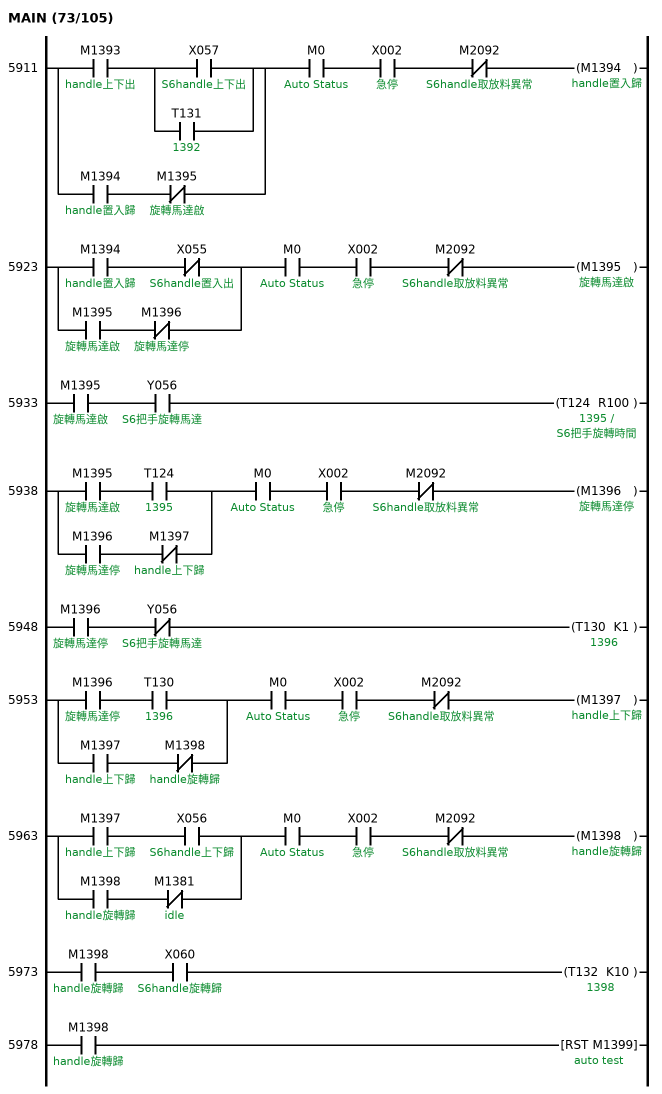
[picture p72: ladder of MAIN, rungs at steps 5911 to 5978]
5911  LD      M1393  ; handle上下出
      LD      X057  ; S6handle上下出
      OR      T131  ; 1392
      ANB
      LD      M1394  ; handle置入歸
      ANI     M1395  ; 旋轉馬達啟
      ORB
      AND     M0  ; Auto Status
      AND     X002  ; 急停
      ANI     M2092  ; S6handle取放料異常
      OUT     M1394  ; handle置入歸
5923  LD      M1394  ; handle置入歸
      ANI     X055  ; S6handle置入出
      LD      M1395  ; 旋轉馬達啟
      ANI     M1396  ; 旋轉馬達停
      ORB
      AND     M0  ; Auto Status
      AND     X002  ; 急停
      ANI     M2092  ; S6handle取放料異常
      OUT     M1395  ; 旋轉馬達啟
5933  LD      M1395  ; 旋轉馬達啟
      AND     Y056  ; S6把手旋轉馬達
      OUT     T124 R100  ; 1395 / S6把手旋轉時間
5938  LD      M1395  ; 旋轉馬達啟
      AND     T124  ; 1395
      LD      M1396  ; 旋轉馬達停
      ANI     M1397  ; handle上下歸
      ORB
      AND     M0  ; Auto Status
      AND     X002  ; 急停
      ANI     M2092  ; S6handle取放料異常
      OUT     M1396  ; 旋轉馬達停
5948  LD      M1396  ; 旋轉馬達停
      ANI     Y056  ; S6把手旋轉馬達
      OUT     T130 K1  ; 1396
5953  LD      M1396  ; 旋轉馬達停
      AND     T130  ; 1396
      LD      M1397  ; handle上下歸
      ANI     M1398  ; handle旋轉歸
      ORB
      AND     M0  ; Auto Status
      AND     X002  ; 急停
      ANI     M2092  ; S6handle取放料異常
      OUT     M1397  ; handle上下歸
5963  LD      M1397  ; handle上下歸
      AND     X056  ; S6handle上下歸
      LD      M1398  ; handle旋轉歸
      ANI     M1381  ; idle
      ORB
      AND     M0  ; Auto Status
      AND     X002  ; 急停
      ANI     M2092  ; S6handle取放料異常
      OUT     M1398  ; handle旋轉歸
5973  LD      M1398  ; handle旋轉歸
      AND     X060  ; S6handle旋轉歸
      OUT     T132 K10  ; 1398
5978  LD      M1398  ; handle旋轉歸
      RST     M1399  ; auto test
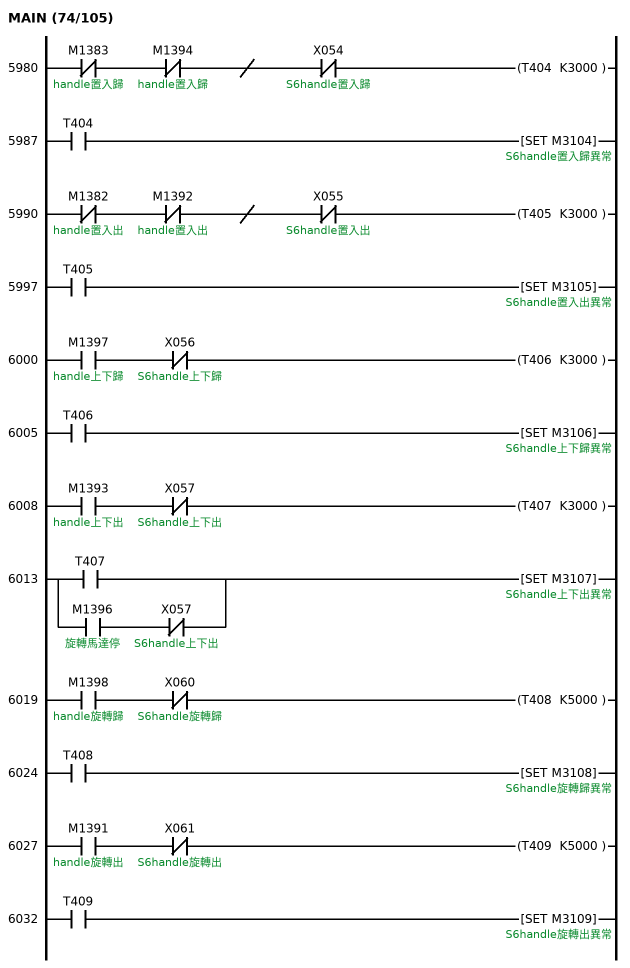
5980  LDI     M1383  ; handle置入歸
      ANI     M1394  ; handle置入歸
      INV
      ANI     X054  ; S6handle置入歸
      OUT     T404 K3000
5987  LD      T404
      SET     M3104  ; S6handle置入歸異常
5990  LDI     M1382  ; handle置入出
      ANI     M1392  ; handle置入出
      INV
      ANI     X055  ; S6handle置入出
      OUT     T405 K3000
5997  LD      T405
      SET     M3105  ; S6handle置入出異常
6000  LD      M1397  ; handle上下歸
      ANI     X056  ; S6handle上下歸
      OUT     T406 K3000
6005  LD      T406
      SET     M3106  ; S6handle上下歸異常
6008  LD      M1393  ; handle上下出
      ANI     X057  ; S6handle上下出
      OUT     T407 K3000
6013  LD      T407
      LD      M1396  ; 旋轉馬達停
      ANI     X057  ; S6handle上下出
      ORB
      SET     M3107  ; S6handle上下出異常
6019  LD      M1398  ; handle旋轉歸
      ANI     X060  ; S6handle旋轉歸
      OUT     T408 K5000
6024  LD      T408
      SET     M3108  ; S6handle旋轉歸異常
6027  LD      M1391  ; handle旋轉出
      ANI     X061  ; S6handle旋轉出
      OUT     T409 K5000
6032  LD      T409
      SET     M3109  ; S6handle旋轉出異常
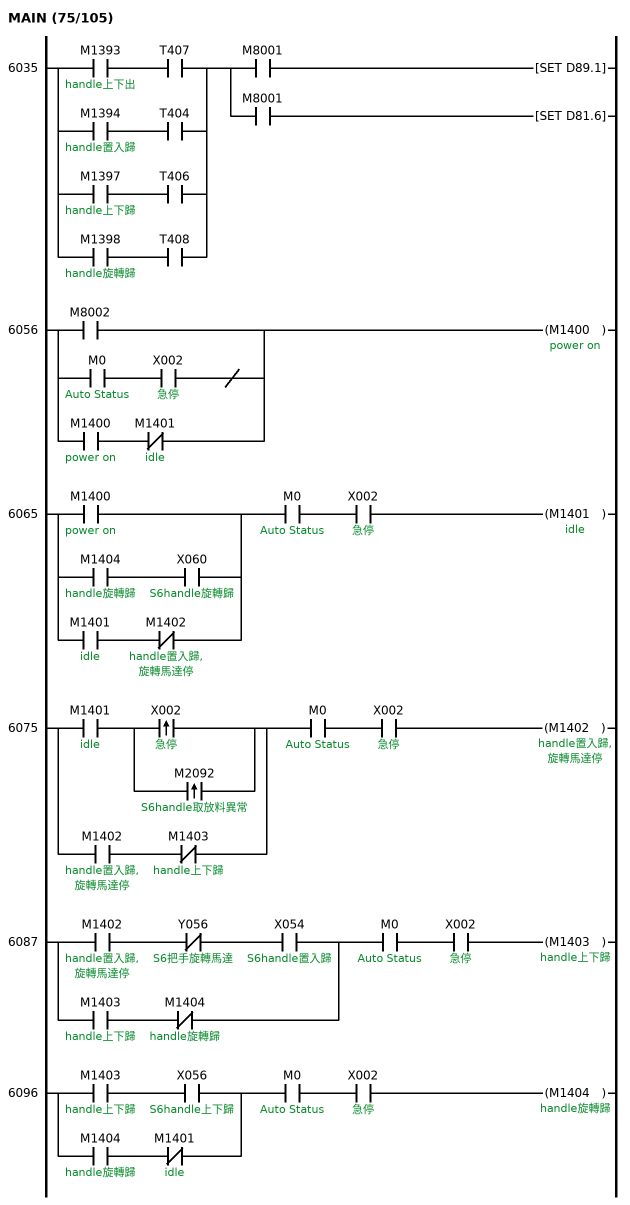
6035  LD      M1393  ; handle上下出
      AND     T407
      LD      M1394  ; handle置入歸
      AND     T404
      ORB
      LD      M1397  ; handle上下歸
      AND     T406
      ORB
      LD      M1398  ; handle旋轉歸
      AND     T408
      ORB
      MPS
      AND     M8001
      SET     D89.1
      MPP
      AND     M8001
      SET     D81.6
6056  LD      M8002
      LD      M0  ; Auto Status
      AND     X002  ; 急停
      INV
      ORB
      LD      M1400  ; power on
      ANI     M1401  ; idle
      ORB
      OUT     M1400  ; power on
6065  LD      M1400  ; power on
      LD      M1404  ; handle旋轉歸
      AND     X060  ; S6handle旋轉歸
      ORB
      LD      M1401  ; idle
      ANI     M1402  ; handle置入歸,旋轉馬達停
      ORB
      AND     M0  ; Auto Status
      AND     X002  ; 急停
      OUT     M1401  ; idle
6075  LD      M1401  ; idle
      LDP     X002  ; 急停
      ORP     M2092  ; S6handle取放料異常
      ANB
      LD      M1402  ; handle置入歸,旋轉馬達停
      ANI     M1403  ; handle上下歸
      ORB
      AND     M0  ; Auto Status
      AND     X002  ; 急停
      OUT     M1402  ; handle置入歸,旋轉馬達停
6087  LD      M1402  ; handle置入歸,旋轉馬達停
      ANI     Y056  ; S6把手旋轉馬達
      AND     X054  ; S6handle置入歸
      LD      M1403  ; handle上下歸
      ANI     M1404  ; handle旋轉歸
      ORB
      AND     M0  ; Auto Status
      AND     X002  ; 急停
      OUT     M1403  ; handle上下歸
6096  LD      M1403  ; handle上下歸
      AND     X056  ; S6handle上下歸
      LD      M1404  ; handle旋轉歸
      ANI     M1401  ; idle
      ORB
      AND     M0  ; Auto Status
      AND     X002  ; 急停
      OUT     M1404  ; handle旋轉歸
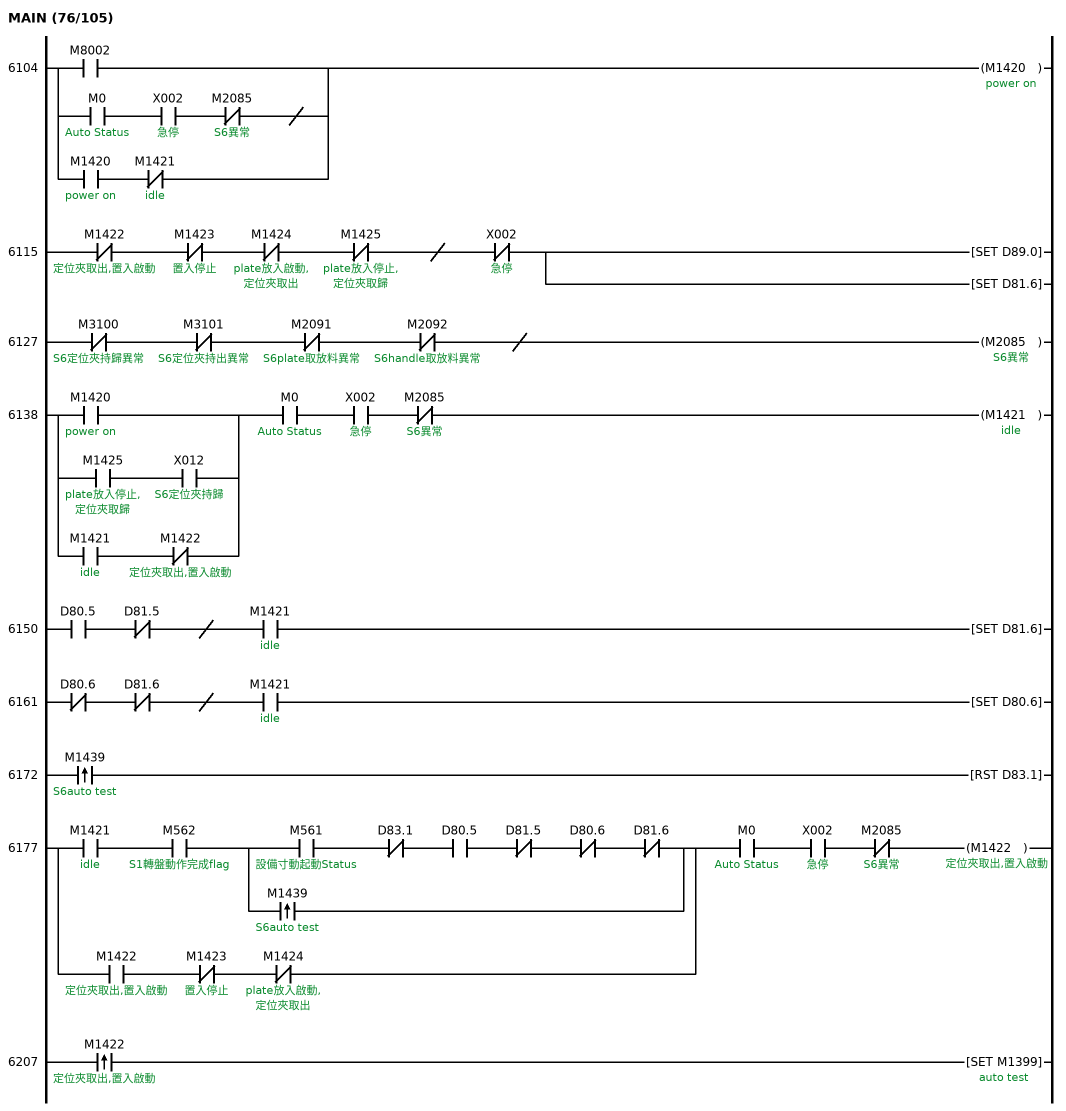
6104  LD      M8002
      LD      M0  ; Auto Status
      AND     X002  ; 急停
      ANI     M2085  ; S6異常
      INV
      ORB
      LD      M1420  ; power on
      ANI     M1421  ; idle
      ORB
      OUT     M1420  ; power on
6115  LDI     M1422  ; 定位夾取出,置入啟動
      ANI     M1423  ; 置入停止
      ANI     M1424  ; plate放入啟動,定位夾取出
      ANI     M1425  ; plate放入停止,定位夾取歸
      INV
      ANI     X002  ; 急停
      SET     D89.0
      SET     D81.6
6127  LDI     M3100  ; S6定位夾持歸異常
      ANI     M3101  ; S6定位夾持出異常
      ANI     M2091  ; S6plate取放料異常
      ANI     M2092  ; S6handle取放料異常
      INV
      OUT     M2085  ; S6異常
6138  LD      M1420  ; power on
      LD      M1425  ; plate放入停止,定位夾取歸
      AND     X012  ; S6定位夾持歸
      ORB
      LD      M1421  ; idle
      ANI     M1422  ; 定位夾取出,置入啟動
      ORB
      AND     M0  ; Auto Status
      AND     X002  ; 急停
      ANI     M2085  ; S6異常
      OUT     M1421  ; idle
6150  LD      D80.5
      ANI     D81.5
      INV
      AND     M1421  ; idle
      SET     D81.6
6161  LDI     D80.6
      ANI     D81.6
      INV
      AND     M1421  ; idle
      SET     D80.6
6172  LDP     M1439  ; S6auto test
      RST     D83.1
6177  LD      M1421  ; idle
      AND     M562  ; S1轉盤動作完成flag
      LD      M561  ; 設備寸動起動Status
      ANI     D83.1
      AND     D80.5
      ANI     D81.5
      ANI     D80.6
      ANI     D81.6
      ORP     M1439  ; S6auto test
      ANB
      LD      M1422  ; 定位夾取出,置入啟動
      ANI     M1423  ; 置入停止
      ANI     M1424  ; plate放入啟動,定位夾取出
      ORB
      AND     M0  ; Auto Status
      AND     X002  ; 急停
      ANI     M2085  ; S6異常
      OUT     M1422  ; 定位夾取出,置入啟動
6207  LDP     M1422  ; 定位夾取出,置入啟動
      SET     M1399  ; auto test
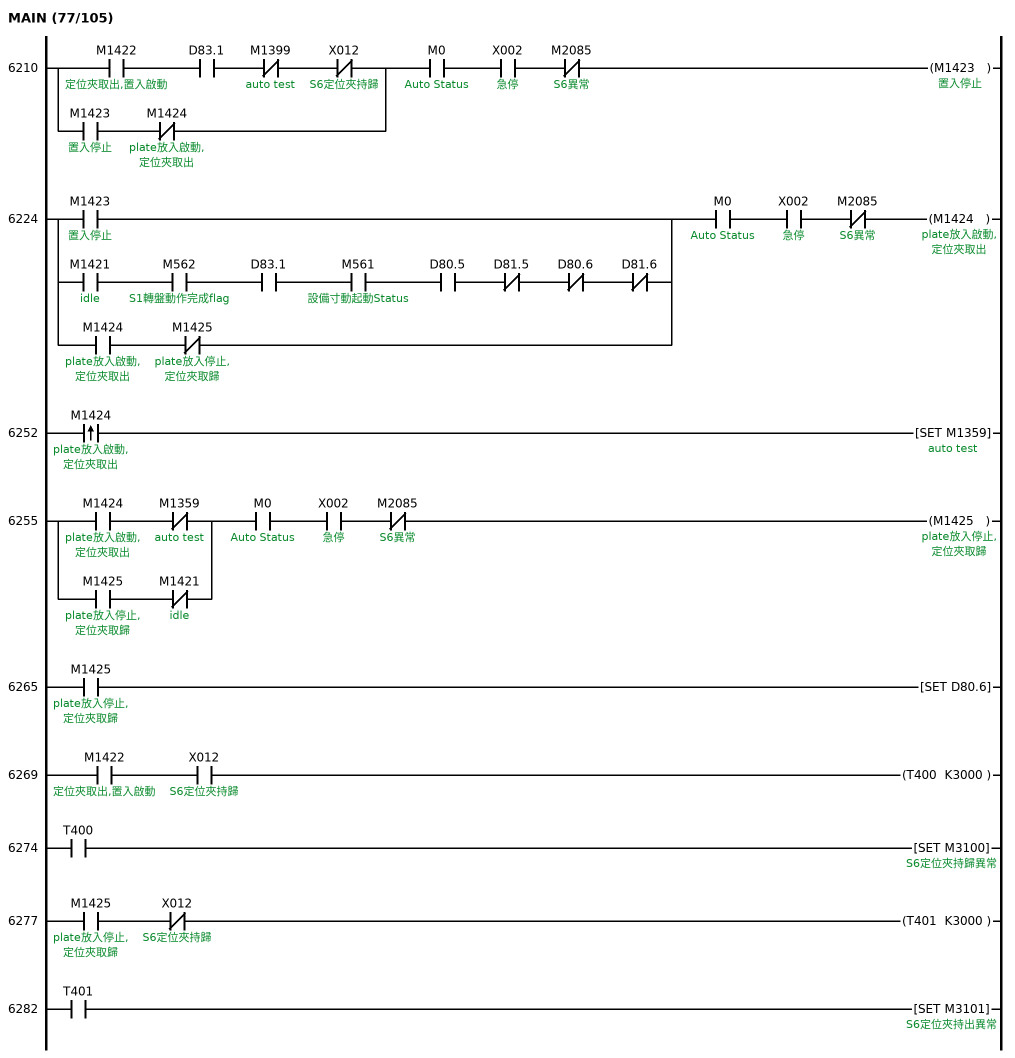
6210  LD      M1422  ; 定位夾取出,置入啟動
      AND     D83.1
      ANI     M1399  ; auto test
      ANI     X012  ; S6定位夾持歸
      LD      M1423  ; 置入停止
      ANI     M1424  ; plate放入啟動,定位夾取出
      ORB
      AND     M0  ; Auto Status
      AND     X002  ; 急停
      ANI     M2085  ; S6異常
      OUT     M1423  ; 置入停止
6224  LD      M1423  ; 置入停止
      LD      M1421  ; idle
      AND     M562  ; S1轉盤動作完成flag
      AND     D83.1
      AND     M561  ; 設備寸動起動Status
      AND     D80.5
      ANI     D81.5
      ANI     D80.6
      ANI     D81.6
      ORB
      LD      M1424  ; plate放入啟動,定位夾取出
      ANI     M1425  ; plate放入停止,定位夾取歸
      ORB
      AND     M0  ; Auto Status
      AND     X002  ; 急停
      ANI     M2085  ; S6異常
      OUT     M1424  ; plate放入啟動,定位夾取出
6252  LDP     M1424  ; plate放入啟動,定位夾取出
      SET     M1359  ; auto test
6255  LD      M1424  ; plate放入啟動,定位夾取出
      ANI     M1359  ; auto test
      LD      M1425  ; plate放入停止,定位夾取歸
      ANI     M1421  ; idle
      ORB
      AND     M0  ; Auto Status
      AND     X002  ; 急停
      ANI     M2085  ; S6異常
      OUT     M1425  ; plate放入停止,定位夾取歸
6265  LD      M1425  ; plate放入停止,定位夾取歸
      SET     D80.6
6269  LD      M1422  ; 定位夾取出,置入啟動
      AND     X012  ; S6定位夾持歸
      OUT     T400 K3000
6274  LD      T400
      SET     M3100  ; S6定位夾持歸異常
6277  LD      M1425  ; plate放入停止,定位夾取歸
      ANI     X012  ; S6定位夾持歸
      OUT     T401 K3000
6282  LD      T401
      SET     M3101  ; S6定位夾持出異常
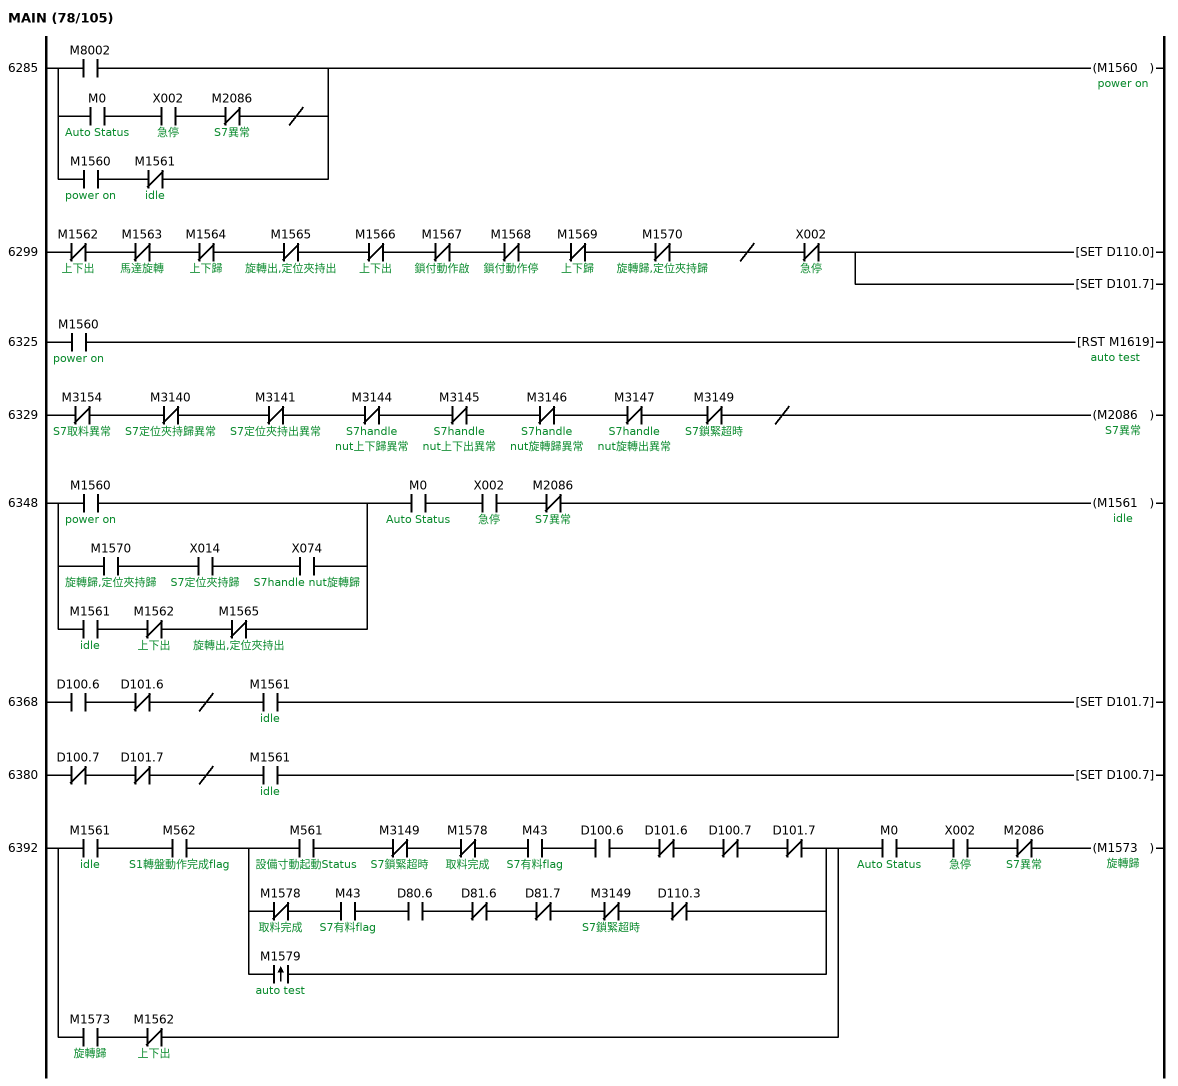
6285  LD      M8002
      LD      M0  ; Auto Status
      AND     X002  ; 急停
      ANI     M2086  ; S7異常
      INV
      ORB
      LD      M1560  ; power on
      ANI     M1561  ; idle
      ORB
      OUT     M1560  ; power on
6299  LDI     M1562  ; 上下出
      ANI     M1563  ; 馬達旋轉
      ANI     M1564  ; 上下歸
      ANI     M1565  ; 旋轉出,定位夾持出
      ANI     M1566  ; 上下出
      ANI     M1567  ; 鎖付動作啟
      ANI     M1568  ; 鎖付動作停
      ANI     M1569  ; 上下歸
      ANI     M1570  ; 旋轉歸,定位夾持歸
      INV
      ANI     X002  ; 急停
      SET     D110.0
      SET     D101.7
6325  LD      M1560  ; power on
      RST     M1619  ; auto test
6329  LDI     M3154  ; S7取料異常
      ANI     M3140  ; S7定位夾持歸異常
      ANI     M3141  ; S7定位夾持出異常
      ANI     M3144  ; S7handle nut上下歸異常
      ANI     M3145  ; S7handle nut上下出異常
      ANI     M3146  ; S7handle nut旋轉歸異常
      ANI     M3147  ; S7handle nut旋轉出異常
      ANI     M3149  ; S7鎖緊超時
      INV
      OUT     M2086  ; S7異常
6348  LD      M1560  ; power on
      LD      M1570  ; 旋轉歸,定位夾持歸
      AND     X014  ; S7定位夾持歸
      AND     X074  ; S7handle nut旋轉歸
      ORB
      LD      M1561  ; idle
      ANI     M1562  ; 上下出
      ANI     M1565  ; 旋轉出,定位夾持出
      ORB
      AND     M0  ; Auto Status
      AND     X002  ; 急停
      ANI     M2086  ; S7異常
      OUT     M1561  ; idle
6368  LD      D100.6
      ANI     D101.6
      INV
      AND     M1561  ; idle
      SET     D101.7
6380  LDI     D100.7
      ANI     D101.7
      INV
      AND     M1561  ; idle
      SET     D100.7
6392  LD      M1561  ; idle
      AND     M562  ; S1轉盤動作完成flag
      LD      M561  ; 設備寸動起動Status
      ANI     M3149  ; S7鎖緊超時
      ANI     M1578  ; 取料完成
      AND     M43  ; S7有料flag
      AND     D100.6
      ANI     D101.6
      ANI     D100.7
      ANI     D101.7
      LDI     M1578  ; 取料完成
      AND     M43  ; S7有料flag
      AND     D80.6
      ANI     D81.6
      ANI     D81.7
      ANI     M3149  ; S7鎖緊超時
      ANI     D110.3
      ORB
      ORP     M1579  ; auto test
      ANB
      LD      M1573  ; 旋轉歸
      ANI     M1562  ; 上下出
      ORB
      AND     M0  ; Auto Status
      AND     X002  ; 急停
      ANI     M2086  ; S7異常
      OUT     M1573  ; 旋轉歸
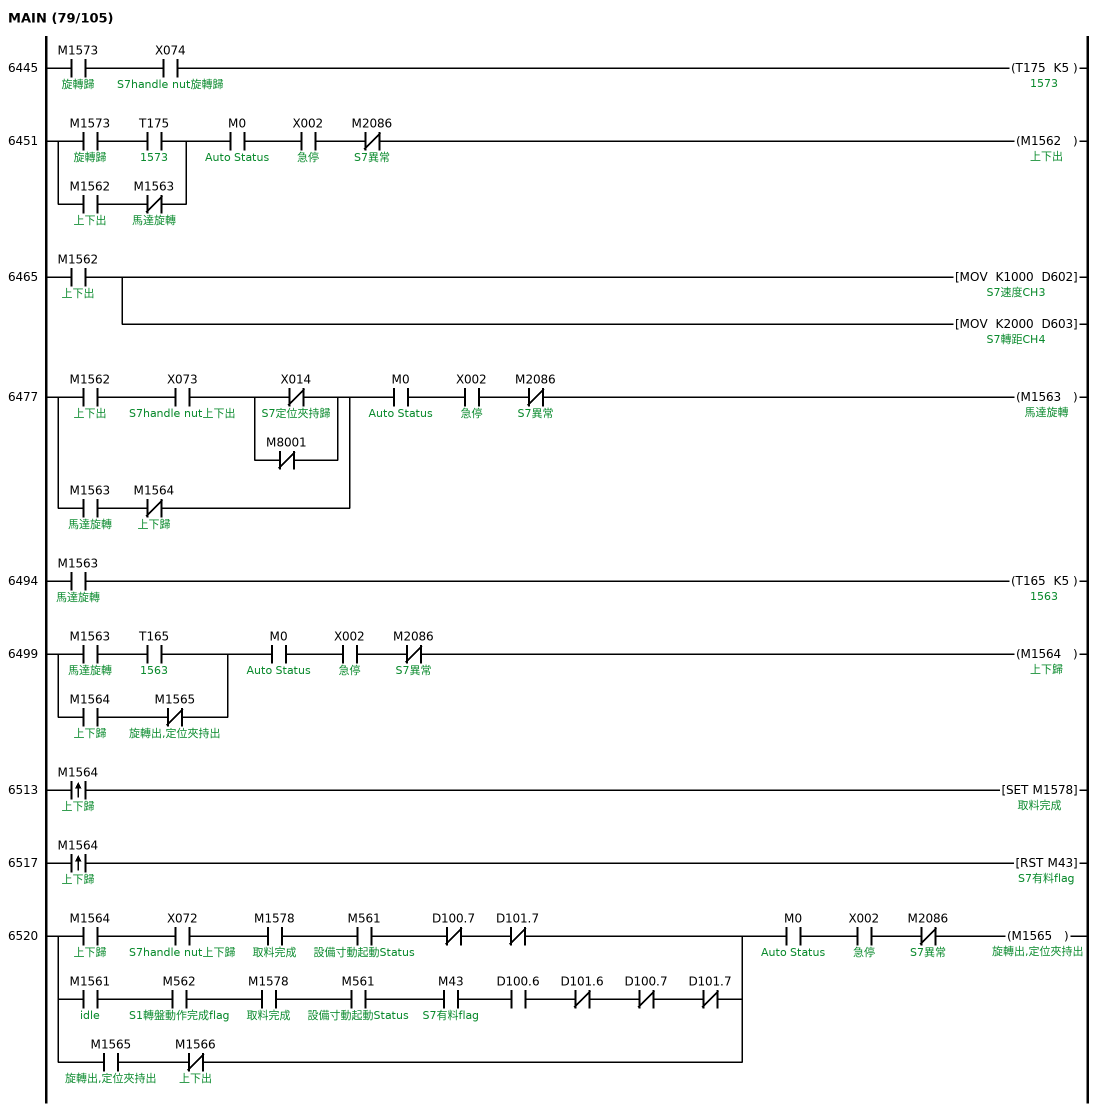
6445  LD      M1573  ; 旋轉歸
      AND     X074  ; S7handle nut旋轉歸
      OUT     T175 K5  ; 1573
6451  LD      M1573  ; 旋轉歸
      AND     T175  ; 1573
      LD      M1562  ; 上下出
      ANI     M1563  ; 馬達旋轉
      ORB
      AND     M0  ; Auto Status
      AND     X002  ; 急停
      ANI     M2086  ; S7異常
      OUT     M1562  ; 上下出
6465  LD      M1562  ; 上下出
      MOV     K1000 D602  ; S7速度CH3
      MOV     K2000 D603  ; S7轉距CH4
6477  LD      M1562  ; 上下出
      AND     X073  ; S7handle nut上下出
      LDI     X014  ; S7定位夾持歸
      ORI     M8001
      ANB
      LD      M1563  ; 馬達旋轉
      ANI     M1564  ; 上下歸
      ORB
      AND     M0  ; Auto Status
      AND     X002  ; 急停
      ANI     M2086  ; S7異常
      OUT     M1563  ; 馬達旋轉
6494  LD      M1563  ; 馬達旋轉
      OUT     T165 K5  ; 1563
6499  LD      M1563  ; 馬達旋轉
      AND     T165  ; 1563
      LD      M1564  ; 上下歸
      ANI     M1565  ; 旋轉出,定位夾持出
      ORB
      AND     M0  ; Auto Status
      AND     X002  ; 急停
      ANI     M2086  ; S7異常
      OUT     M1564  ; 上下歸
6513  LDP     M1564  ; 上下歸
      SET     M1578  ; 取料完成
6517  LDP     M1564  ; 上下歸
      RST     M43  ; S7有料flag
6520  LD      M1564  ; 上下歸
      AND     X072  ; S7handle nut上下歸
      AND     M1578  ; 取料完成
      AND     M561  ; 設備寸動起動Status
      ANI     D100.7
      ANI     D101.7
      LD      M1561  ; idle
      AND     M562  ; S1轉盤動作完成flag
      AND     M1578  ; 取料完成
      AND     M561  ; 設備寸動起動Status
      AND     M43  ; S7有料flag
      AND     D100.6
      ANI     D101.6
      ANI     D100.7
      ANI     D101.7
      ORB
      LD      M1565  ; 旋轉出,定位夾持出
      ANI     M1566  ; 上下出
      ORB
      AND     M0  ; Auto Status
      AND     X002  ; 急停
      ANI     M2086  ; S7異常
      OUT     M1565  ; 旋轉出,定位夾持出
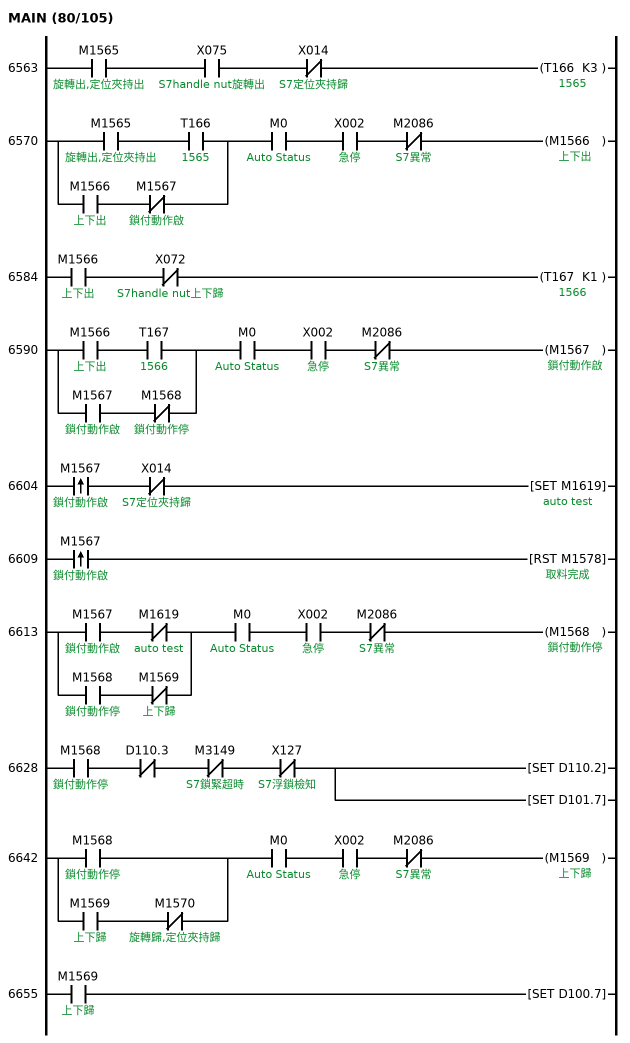
6563  LD      M1565  ; 旋轉出,定位夾持出
      AND     X075  ; S7handle nut旋轉出
      ANI     X014  ; S7定位夾持歸
      OUT     T166 K3  ; 1565
6570  LD      M1565  ; 旋轉出,定位夾持出
      AND     T166  ; 1565
      LD      M1566  ; 上下出
      ANI     M1567  ; 鎖付動作啟
      ORB
      AND     M0  ; Auto Status
      AND     X002  ; 急停
      ANI     M2086  ; S7異常
      OUT     M1566  ; 上下出
6584  LD      M1566  ; 上下出
      ANI     X072  ; S7handle nut上下歸
      OUT     T167 K1  ; 1566
6590  LD      M1566  ; 上下出
      AND     T167  ; 1566
      LD      M1567  ; 鎖付動作啟
      ANI     M1568  ; 鎖付動作停
      ORB
      AND     M0  ; Auto Status
      AND     X002  ; 急停
      ANI     M2086  ; S7異常
      OUT     M1567  ; 鎖付動作啟
6604  LDP     M1567  ; 鎖付動作啟
      ANI     X014  ; S7定位夾持歸
      SET     M1619  ; auto test
6609  LDP     M1567  ; 鎖付動作啟
      RST     M1578  ; 取料完成
6613  LD      M1567  ; 鎖付動作啟
      ANI     M1619  ; auto test
      LD      M1568  ; 鎖付動作停
      ANI     M1569  ; 上下歸
      ORB
      AND     M0  ; Auto Status
      AND     X002  ; 急停
      ANI     M2086  ; S7異常
      OUT     M1568  ; 鎖付動作停
6628  LD      M1568  ; 鎖付動作停
      ANI     D110.3
      ANI     M3149  ; S7鎖緊超時
      ANI     X127  ; S7浮鎖檢知
      SET     D110.2
      SET     D101.7
6642  LD      M1568  ; 鎖付動作停
      LD      M1569  ; 上下歸
      ANI     M1570  ; 旋轉歸,定位夾持歸
      ORB
      AND     M0  ; Auto Status
      AND     X002  ; 急停
      ANI     M2086  ; S7異常
      OUT     M1569  ; 上下歸
6655  LD      M1569  ; 上下歸
      SET     D100.7
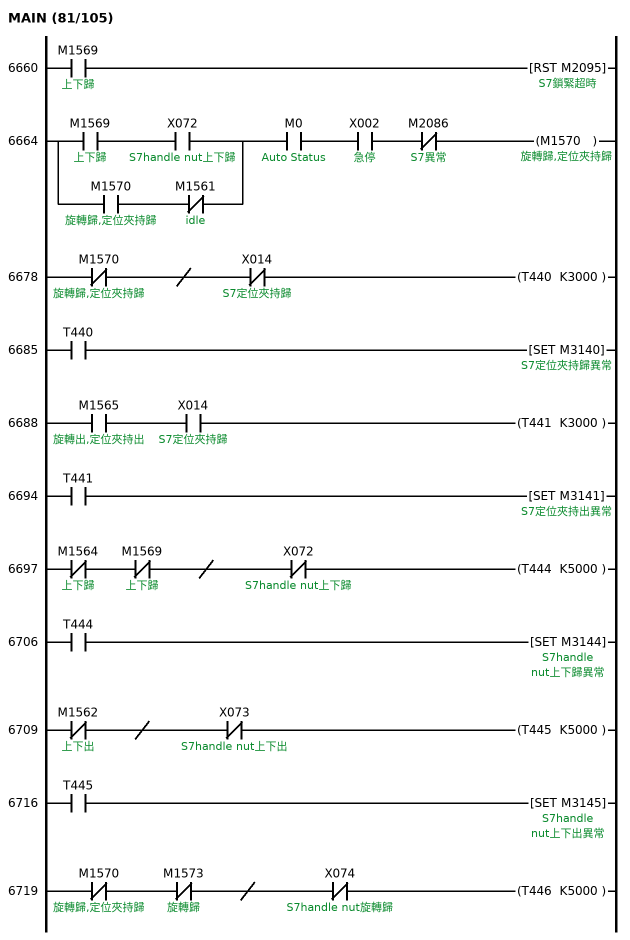
6660  LD      M1569  ; 上下歸
      RST     M2095  ; S7鎖緊超時
6664  LD      M1569  ; 上下歸
      AND     X072  ; S7handle nut上下歸
      LD      M1570  ; 旋轉歸,定位夾持歸
      ANI     M1561  ; idle
      ORB
      AND     M0  ; Auto Status
      AND     X002  ; 急停
      ANI     M2086  ; S7異常
      OUT     M1570  ; 旋轉歸,定位夾持歸
6678  LDI     M1570  ; 旋轉歸,定位夾持歸
      INV
      ANI     X014  ; S7定位夾持歸
      OUT     T440 K3000
6685  LD      T440
      SET     M3140  ; S7定位夾持歸異常
6688  LD      M1565  ; 旋轉出,定位夾持出
      AND     X014  ; S7定位夾持歸
      OUT     T441 K3000
6694  LD      T441
      SET     M3141  ; S7定位夾持出異常
6697  LDI     M1564  ; 上下歸
      ANI     M1569  ; 上下歸
      INV
      ANI     X072  ; S7handle nut上下歸
      OUT     T444 K5000
6706  LD      T444
      SET     M3144  ; S7handle nut上下歸異常
6709  LDI     M1562  ; 上下出
      INV
      ANI     X073  ; S7handle nut上下出
      OUT     T445 K5000
6716  LD      T445
      SET     M3145  ; S7handle nut上下出異常
6719  LDI     M1570  ; 旋轉歸,定位夾持歸
      ANI     M1573  ; 旋轉歸
      INV
      ANI     X074  ; S7handle nut旋轉歸
      OUT     T446 K5000
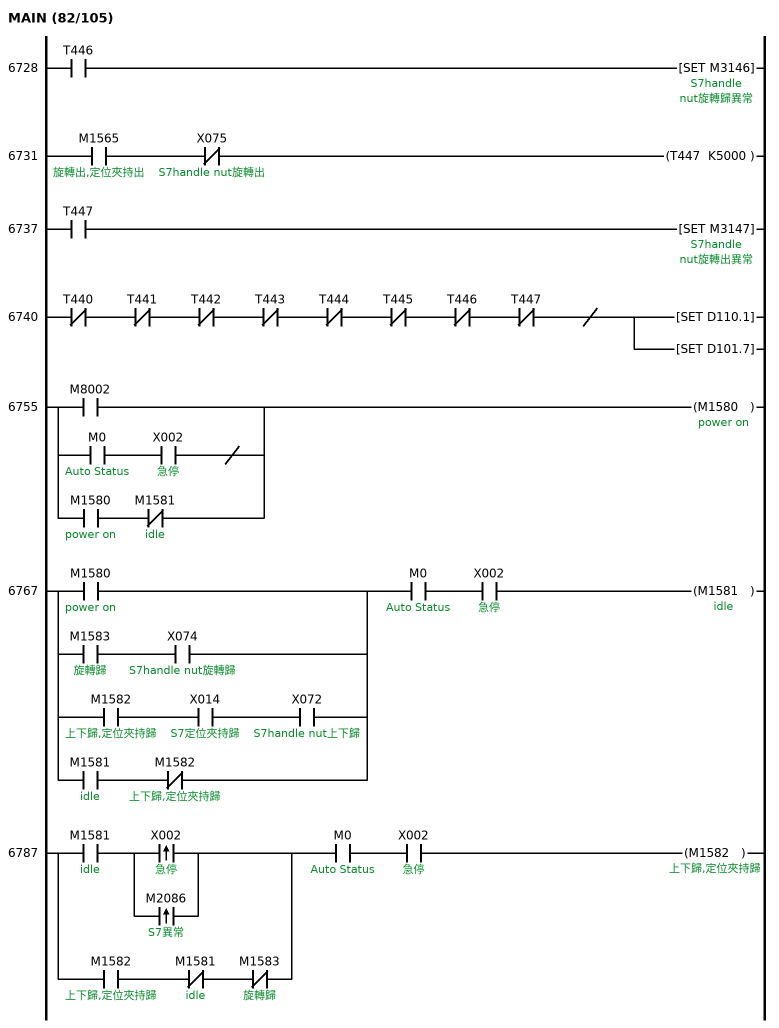
6728  LD      T446
      SET     M3146  ; S7handle nut旋轉歸異常
6731  LD      M1565  ; 旋轉出,定位夾持出
      ANI     X075  ; S7handle nut旋轉出
      OUT     T447 K5000
6737  LD      T447
      SET     M3147  ; S7handle nut旋轉出異常
6740  LDI     T440
      ANI     T441
      ANI     T442
      ANI     T443
      ANI     T444
      ANI     T445
      ANI     T446
      ANI     T447
      INV
      SET     D110.1
      SET     D101.7
6755  LD      M8002
      LD      M0  ; Auto Status
      AND     X002  ; 急停
      INV
      ORB
      LD      M1580  ; power on
      ANI     M1581  ; idle
      ORB
      OUT     M1580  ; power on
6767  LD      M1580  ; power on
      LD      M1583  ; 旋轉歸
      AND     X074  ; S7handle nut旋轉歸
      ORB
      LD      M1582  ; 上下歸,定位夾持歸
      AND     X014  ; S7定位夾持歸
      AND     X072  ; S7handle nut上下歸
      ORB
      LD      M1581  ; idle
      ANI     M1582  ; 上下歸,定位夾持歸
      ORB
      AND     M0  ; Auto Status
      AND     X002  ; 急停
      OUT     M1581  ; idle
6787  LD      M1581  ; idle
      LDP     X002  ; 急停
      ORP     M2086  ; S7異常
      ANB
      LD      M1582  ; 上下歸,定位夾持歸
      ANI     M1581  ; idle
      ANI     M1583  ; 旋轉歸
      ORB
      AND     M0  ; Auto Status
      AND     X002  ; 急停
      OUT     M1582  ; 上下歸,定位夾持歸
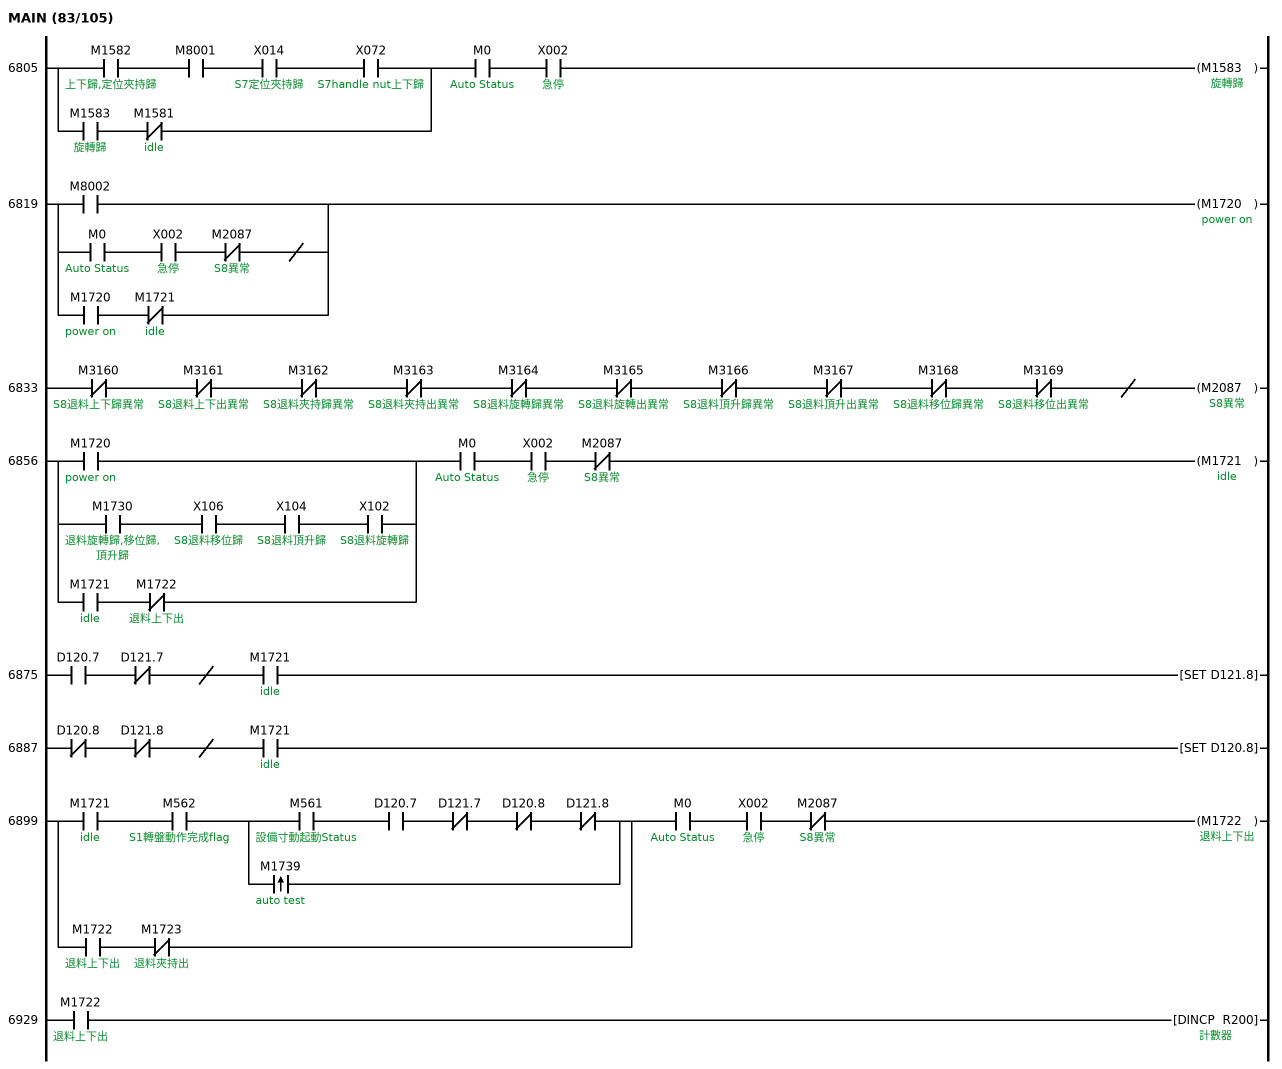
6805  LD      M1582  ; 上下歸,定位夾持歸
      AND     M8001
      AND     X014  ; S7定位夾持歸
      AND     X072  ; S7handle nut上下歸
      LD      M1583  ; 旋轉歸
      ANI     M1581  ; idle
      ORB
      AND     M0  ; Auto Status
      AND     X002  ; 急停
      OUT     M1583  ; 旋轉歸
6819  LD      M8002
      LD      M0  ; Auto Status
      AND     X002  ; 急停
      ANI     M2087  ; S8異常
      INV
      ORB
      LD      M1720  ; power on
      ANI     M1721  ; idle
      ORB
      OUT     M1720  ; power on
6833  LDI     M3160  ; S8退料上下歸異常
      ANI     M3161  ; S8退料上下出異常
      ANI     M3162  ; S8退料夾持歸異常
      ANI     M3163  ; S8退料夾持出異常
      ANI     M3164  ; S8退料旋轉歸異常
      ANI     M3165  ; S8退料旋轉出異常
      ANI     M3166  ; S8退料頂升歸異常
      ANI     M3167  ; S8退料頂升出異常
      ANI     M3168  ; S8退料移位歸異常
      ANI     M3169  ; S8退料移位出異常
      INV
      OUT     M2087  ; S8異常
6856  LD      M1720  ; power on
      LD      M1730  ; 退料旋轉歸,移位歸,頂升歸
      AND     X106  ; S8退料移位歸
      AND     X104  ; S8退料頂升歸
      AND     X102  ; S8退料旋轉歸
      ORB
      LD      M1721  ; idle
      ANI     M1722  ; 退料上下出
      ORB
      AND     M0  ; Auto Status
      AND     X002  ; 急停
      ANI     M2087  ; S8異常
      OUT     M1721  ; idle
6875  LD      D120.7
      ANI     D121.7
      INV
      AND     M1721  ; idle
      SET     D121.8
6887  LDI     D120.8
      ANI     D121.8
      INV
      AND     M1721  ; idle
      SET     D120.8
6899  LD      M1721  ; idle
      AND     M562  ; S1轉盤動作完成flag
      LD      M561  ; 設備寸動起動Status
      AND     D120.7
      ANI     D121.7
      ANI     D120.8
      ANI     D121.8
      ORP     M1739  ; auto test
      ANB
      LD      M1722  ; 退料上下出
      ANI     M1723  ; 退料夾持出
      ORB
      AND     M0  ; Auto Status
      AND     X002  ; 急停
      ANI     M2087  ; S8異常
      OUT     M1722  ; 退料上下出
6929  LD      M1722  ; 退料上下出
      DINCP   R200  ; 計數器
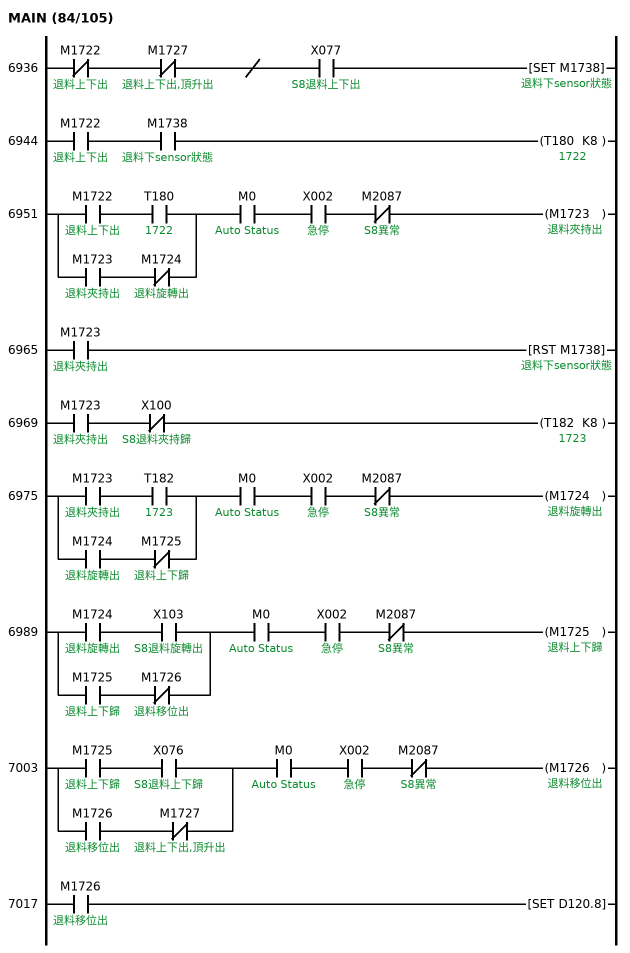
6936  LDI     M1722  ; 退料上下出
      ANI     M1727  ; 退料上下出,頂升出
      INV
      AND     X077  ; S8退料上下出
      SET     M1738  ; 退料下sensor狀態
6944  LD      M1722  ; 退料上下出
      AND     M1738  ; 退料下sensor狀態
      OUT     T180 K8  ; 1722
6951  LD      M1722  ; 退料上下出
      AND     T180  ; 1722
      LD      M1723  ; 退料夾持出
      ANI     M1724  ; 退料旋轉出
      ORB
      AND     M0  ; Auto Status
      AND     X002  ; 急停
      ANI     M2087  ; S8異常
      OUT     M1723  ; 退料夾持出
6965  LD      M1723  ; 退料夾持出
      RST     M1738  ; 退料下sensor狀態
6969  LD      M1723  ; 退料夾持出
      ANI     X100  ; S8退料夾持歸
      OUT     T182 K8  ; 1723
6975  LD      M1723  ; 退料夾持出
      AND     T182  ; 1723
      LD      M1724  ; 退料旋轉出
      ANI     M1725  ; 退料上下歸
      ORB
      AND     M0  ; Auto Status
      AND     X002  ; 急停
      ANI     M2087  ; S8異常
      OUT     M1724  ; 退料旋轉出
6989  LD      M1724  ; 退料旋轉出
      AND     X103  ; S8退料旋轉出
      LD      M1725  ; 退料上下歸
      ANI     M1726  ; 退料移位出
      ORB
      AND     M0  ; Auto Status
      AND     X002  ; 急停
      ANI     M2087  ; S8異常
      OUT     M1725  ; 退料上下歸
7003  LD      M1725  ; 退料上下歸
      AND     X076  ; S8退料上下歸
      LD      M1726  ; 退料移位出
      ANI     M1727  ; 退料上下出,頂升出
      ORB
      AND     M0  ; Auto Status
      AND     X002  ; 急停
      ANI     M2087  ; S8異常
      OUT     M1726  ; 退料移位出
7017  LD      M1726  ; 退料移位出
      SET     D120.8
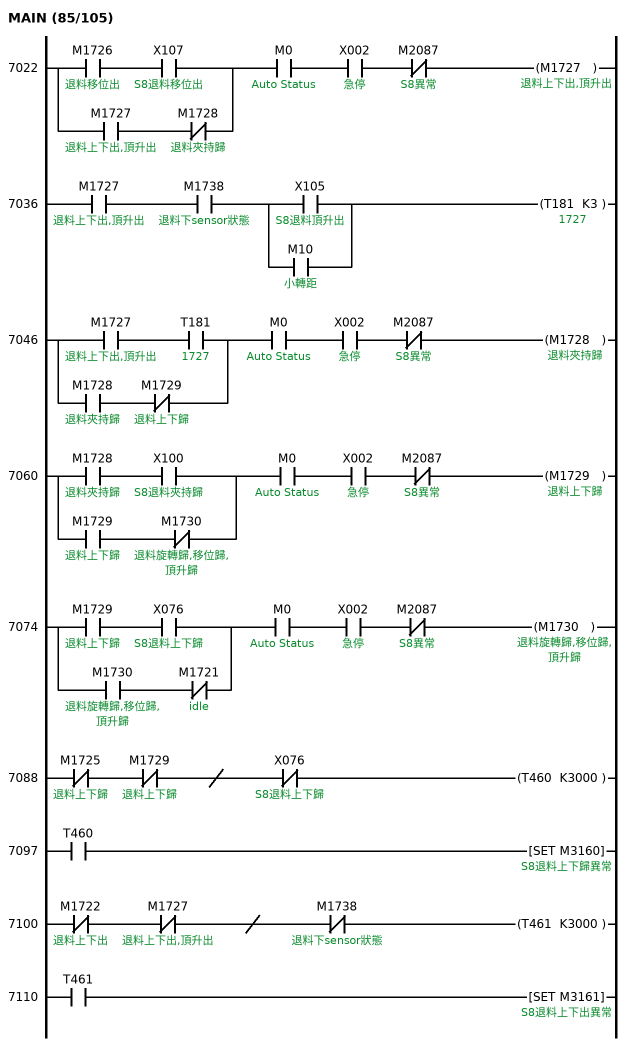
7022  LD      M1726  ; 退料移位出
      AND     X107  ; S8退料移位出
      LD      M1727  ; 退料上下出,頂升出
      ANI     M1728  ; 退料夾持歸
      ORB
      AND     M0  ; Auto Status
      AND     X002  ; 急停
      ANI     M2087  ; S8異常
      OUT     M1727  ; 退料上下出,頂升出
7036  LD      M1727  ; 退料上下出,頂升出
      AND     M1738  ; 退料下sensor狀態
      LD      X105  ; S8退料頂升出
      OR      M10  ; 小轉距
      ANB
      OUT     T181 K3  ; 1727
7046  LD      M1727  ; 退料上下出,頂升出
      AND     T181  ; 1727
      LD      M1728  ; 退料夾持歸
      ANI     M1729  ; 退料上下歸
      ORB
      AND     M0  ; Auto Status
      AND     X002  ; 急停
      ANI     M2087  ; S8異常
      OUT     M1728  ; 退料夾持歸
7060  LD      M1728  ; 退料夾持歸
      AND     X100  ; S8退料夾持歸
      LD      M1729  ; 退料上下歸
      ANI     M1730  ; 退料旋轉歸,移位歸,頂升歸
      ORB
      AND     M0  ; Auto Status
      AND     X002  ; 急停
      ANI     M2087  ; S8異常
      OUT     M1729  ; 退料上下歸
7074  LD      M1729  ; 退料上下歸
      AND     X076  ; S8退料上下歸
      LD      M1730  ; 退料旋轉歸,移位歸,頂升歸
      ANI     M1721  ; idle
      ORB
      AND     M0  ; Auto Status
      AND     X002  ; 急停
      ANI     M2087  ; S8異常
      OUT     M1730  ; 退料旋轉歸,移位歸,頂升歸
7088  LDI     M1725  ; 退料上下歸
      ANI     M1729  ; 退料上下歸
      INV
      ANI     X076  ; S8退料上下歸
      OUT     T460 K3000
7097  LD      T460
      SET     M3160  ; S8退料上下歸異常
7100  LDI     M1722  ; 退料上下出
      ANI     M1727  ; 退料上下出,頂升出
      INV
      ANI     M1738  ; 退料下sensor狀態
      OUT     T461 K3000
7110  LD      T461
      SET     M3161  ; S8退料上下出異常
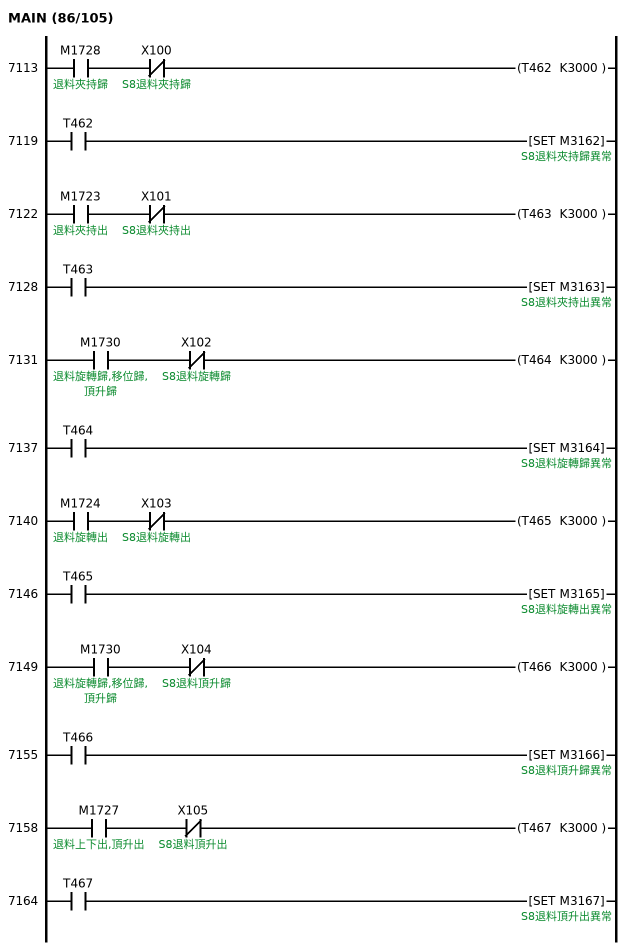
7113  LD      M1728  ; 退料夾持歸
      ANI     X100  ; S8退料夾持歸
      OUT     T462 K3000
7119  LD      T462
      SET     M3162  ; S8退料夾持歸異常
7122  LD      M1723  ; 退料夾持出
      ANI     X101  ; S8退料夾持出
      OUT     T463 K3000
7128  LD      T463
      SET     M3163  ; S8退料夾持出異常
7131  LD      M1730  ; 退料旋轉歸,移位歸,頂升歸
      ANI     X102  ; S8退料旋轉歸
      OUT     T464 K3000
7137  LD      T464
      SET     M3164  ; S8退料旋轉歸異常
7140  LD      M1724  ; 退料旋轉出
      ANI     X103  ; S8退料旋轉出
      OUT     T465 K3000
7146  LD      T465
      SET     M3165  ; S8退料旋轉出異常
7149  LD      M1730  ; 退料旋轉歸,移位歸,頂升歸
      ANI     X104  ; S8退料頂升歸
      OUT     T466 K3000
7155  LD      T466
      SET     M3166  ; S8退料頂升歸異常
7158  LD      M1727  ; 退料上下出,頂升出
      ANI     X105  ; S8退料頂升出
      OUT     T467 K3000
7164  LD      T467
      SET     M3167  ; S8退料頂升出異常
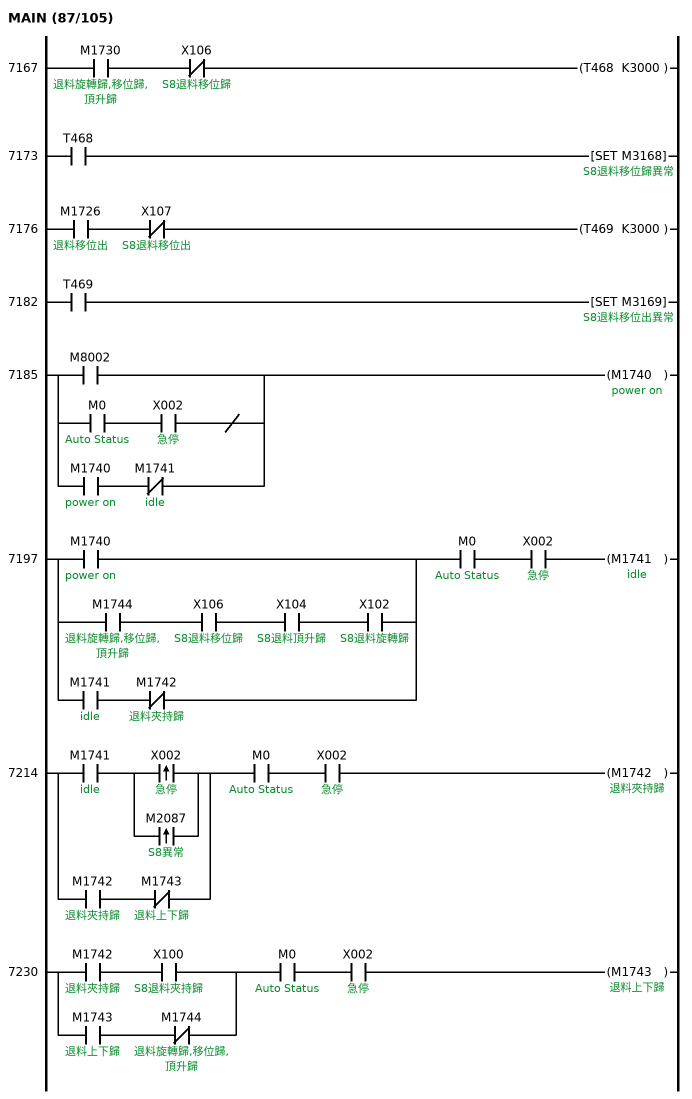
7167  LD      M1730  ; 退料旋轉歸,移位歸,頂升歸
      ANI     X106  ; S8退料移位歸
      OUT     T468 K3000
7173  LD      T468
      SET     M3168  ; S8退料移位歸異常
7176  LD      M1726  ; 退料移位出
      ANI     X107  ; S8退料移位出
      OUT     T469 K3000
7182  LD      T469
      SET     M3169  ; S8退料移位出異常
7185  LD      M8002
      LD      M0  ; Auto Status
      AND     X002  ; 急停
      INV
      ORB
      LD      M1740  ; power on
      ANI     M1741  ; idle
      ORB
      OUT     M1740  ; power on
7197  LD      M1740  ; power on
      LD      M1744  ; 退料旋轉歸,移位歸,頂升歸
      AND     X106  ; S8退料移位歸
      AND     X104  ; S8退料頂升歸
      AND     X102  ; S8退料旋轉歸
      ORB
      LD      M1741  ; idle
      ANI     M1742  ; 退料夾持歸
      ORB
      AND     M0  ; Auto Status
      AND     X002  ; 急停
      OUT     M1741  ; idle
7214  LD      M1741  ; idle
      LDP     X002  ; 急停
      ORP     M2087  ; S8異常
      ANB
      LD      M1742  ; 退料夾持歸
      ANI     M1743  ; 退料上下歸
      ORB
      AND     M0  ; Auto Status
      AND     X002  ; 急停
      OUT     M1742  ; 退料夾持歸
7230  LD      M1742  ; 退料夾持歸
      AND     X100  ; S8退料夾持歸
      LD      M1743  ; 退料上下歸
      ANI     M1744  ; 退料旋轉歸,移位歸,頂升歸
      ORB
      AND     M0  ; Auto Status
      AND     X002  ; 急停
      OUT     M1743  ; 退料上下歸
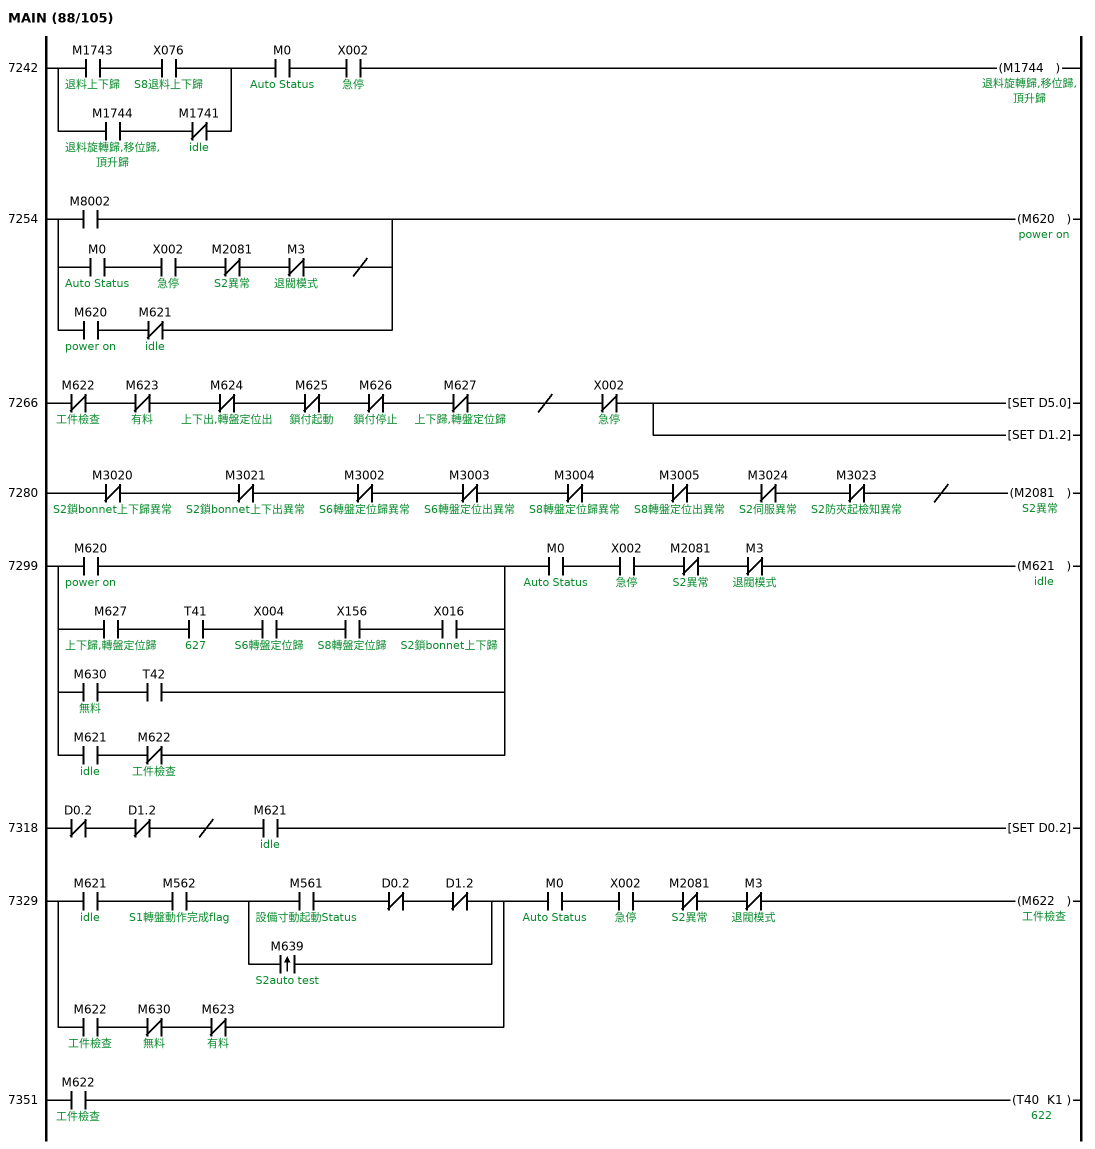
7242  LD      M1743  ; 退料上下歸
      AND     X076  ; S8退料上下歸
      LD      M1744  ; 退料旋轉歸,移位歸,頂升歸
      ANI     M1741  ; idle
      ORB
      AND     M0  ; Auto Status
      AND     X002  ; 急停
      OUT     M1744  ; 退料旋轉歸,移位歸,頂升歸
7254  LD      M8002
      LD      M0  ; Auto Status
      AND     X002  ; 急停
      ANI     M2081  ; S2異常
      ANI     M3  ; 退閥模式
      INV
      ORB
      LD      M620  ; power on
      ANI     M621  ; idle
      ORB
      OUT     M620  ; power on
7266  LDI     M622  ; 工件檢查
      ANI     M623  ; 有料
      ANI     M624  ; 上下出,轉盤定位出
      ANI     M625  ; 鎖付起動
      ANI     M626  ; 鎖付停止
      ANI     M627  ; 上下歸,轉盤定位歸
      INV
      ANI     X002  ; 急停
      SET     D5.0
      SET     D1.2
7280  LDI     M3020  ; S2鎖bonnet上下歸異常
      ANI     M3021  ; S2鎖bonnet上下出異常
      ANI     M3002  ; S6轉盤定位歸異常
      ANI     M3003  ; S6轉盤定位出異常
      ANI     M3004  ; S8轉盤定位歸異常
      ANI     M3005  ; S8轉盤定位出異常
      ANI     M3024  ; S2伺服異常
      ANI     M3023  ; S2防夾起檢知異常
      INV
      OUT     M2081  ; S2異常
7299  LD      M620  ; power on
      LD      M627  ; 上下歸,轉盤定位歸
      AND     T41  ; 627
      AND     X004  ; S6轉盤定位歸
      AND     X156  ; S8轉盤定位歸
      AND     X016  ; S2鎖bonnet上下歸
      ORB
      LD      M630  ; 無料
      AND     T42
      ORB
      LD      M621  ; idle
      ANI     M622  ; 工件檢查
      ORB
      AND     M0  ; Auto Status
      AND     X002  ; 急停
      ANI     M2081  ; S2異常
      ANI     M3  ; 退閥模式
      OUT     M621  ; idle
7318  LDI     D0.2
      ANI     D1.2
      INV
      AND     M621  ; idle
      SET     D0.2
7329  LD      M621  ; idle
      AND     M562  ; S1轉盤動作完成flag
      LD      M561  ; 設備寸動起動Status
      ANI     D0.2
      ANI     D1.2
      ORP     M639  ; S2auto test
      ANB
      LD      M622  ; 工件檢查
      ANI     M630  ; 無料
      ANI     M623  ; 有料
      ORB
      AND     M0  ; Auto Status
      AND     X002  ; 急停
      ANI     M2081  ; S2異常
      ANI     M3  ; 退閥模式
      OUT     M622  ; 工件檢查
7351  LD      M622  ; 工件檢查
      OUT     T40 K1  ; 622
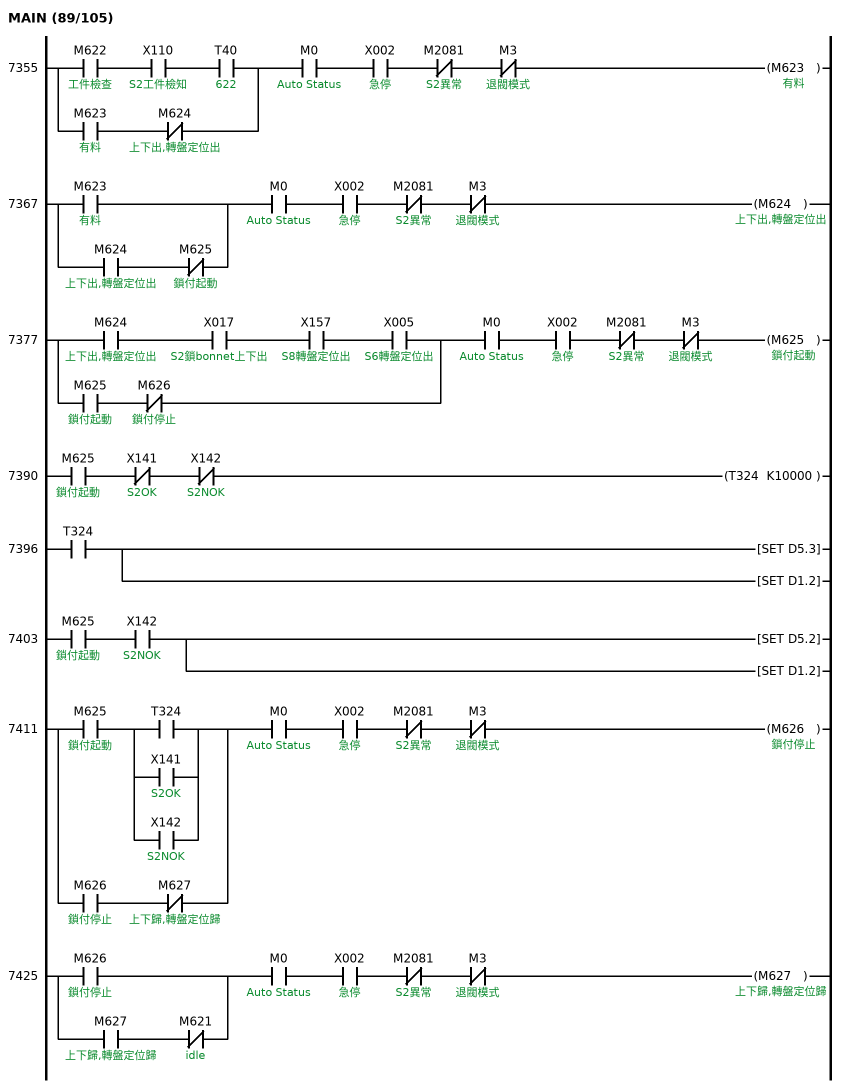
7355  LD      M622  ; 工件檢查
      AND     X110  ; S2工件檢知
      AND     T40  ; 622
      LD      M623  ; 有料
      ANI     M624  ; 上下出,轉盤定位出
      ORB
      AND     M0  ; Auto Status
      AND     X002  ; 急停
      ANI     M2081  ; S2異常
      ANI     M3  ; 退閥模式
      OUT     M623  ; 有料
7367  LD      M623  ; 有料
      LD      M624  ; 上下出,轉盤定位出
      ANI     M625  ; 鎖付起動
      ORB
      AND     M0  ; Auto Status
      AND     X002  ; 急停
      ANI     M2081  ; S2異常
      ANI     M3  ; 退閥模式
      OUT     M624  ; 上下出,轉盤定位出
7377  LD      M624  ; 上下出,轉盤定位出
      AND     X017  ; S2鎖bonnet上下出
      AND     X157  ; S8轉盤定位出
      AND     X005  ; S6轉盤定位出
      LD      M625  ; 鎖付起動
      ANI     M626  ; 鎖付停止
      ORB
      AND     M0  ; Auto Status
      AND     X002  ; 急停
      ANI     M2081  ; S2異常
      ANI     M3  ; 退閥模式
      OUT     M625  ; 鎖付起動
7390  LD      M625  ; 鎖付起動
      ANI     X141  ; S2OK
      ANI     X142  ; S2NOK
      OUT     T324 K10000
7396  LD      T324
      SET     D5.3
      SET     D1.2
7403  LD      M625  ; 鎖付起動
      AND     X142  ; S2NOK
      SET     D5.2
      SET     D1.2
7411  LD      M625  ; 鎖付起動
      LD      T324
      OR      X141  ; S2OK
      OR      X142  ; S2NOK
      ANB
      LD      M626  ; 鎖付停止
      ANI     M627  ; 上下歸,轉盤定位歸
      ORB
      AND     M0  ; Auto Status
      AND     X002  ; 急停
      ANI     M2081  ; S2異常
      ANI     M3  ; 退閥模式
      OUT     M626  ; 鎖付停止
7425  LD      M626  ; 鎖付停止
      LD      M627  ; 上下歸,轉盤定位歸
      ANI     M621  ; idle
      ORB
      AND     M0  ; Auto Status
      AND     X002  ; 急停
      ANI     M2081  ; S2異常
      ANI     M3  ; 退閥模式
      OUT     M627  ; 上下歸,轉盤定位歸
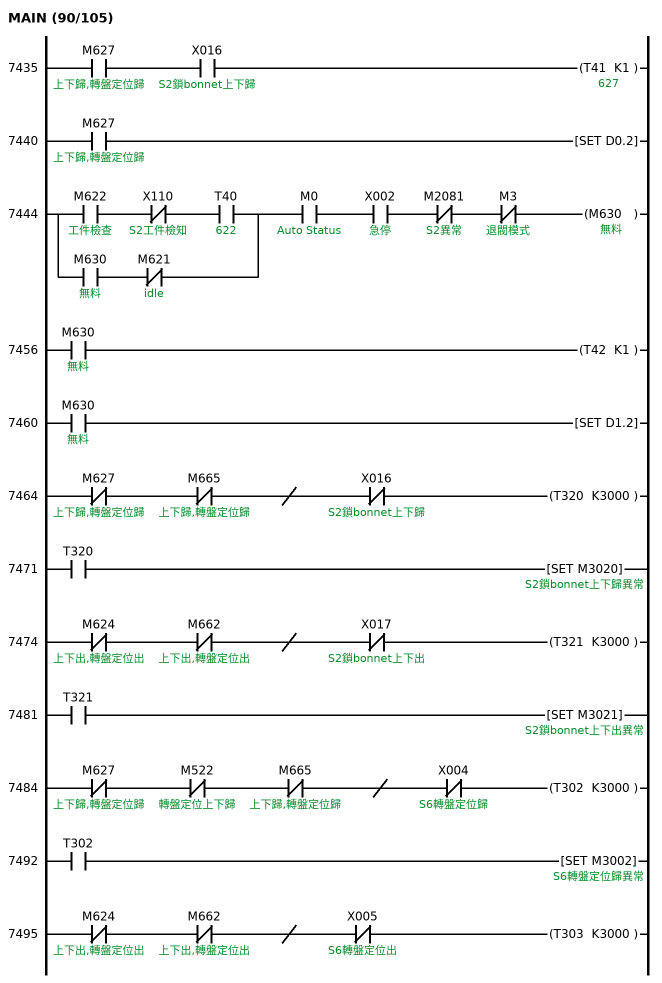
7435  LD      M627  ; 上下歸,轉盤定位歸
      AND     X016  ; S2鎖bonnet上下歸
      OUT     T41 K1  ; 627
7440  LD      M627  ; 上下歸,轉盤定位歸
      SET     D0.2
7444  LD      M622  ; 工件檢查
      ANI     X110  ; S2工件檢知
      AND     T40  ; 622
      LD      M630  ; 無料
      ANI     M621  ; idle
      ORB
      AND     M0  ; Auto Status
      AND     X002  ; 急停
      ANI     M2081  ; S2異常
      ANI     M3  ; 退閥模式
      OUT     M630  ; 無料
7456  LD      M630  ; 無料
      OUT     T42 K1
7460  LD      M630  ; 無料
      SET     D1.2
7464  LDI     M627  ; 上下歸,轉盤定位歸
      ANI     M665  ; 上下歸,轉盤定位歸
      INV
      ANI     X016  ; S2鎖bonnet上下歸
      OUT     T320 K3000
7471  LD      T320
      SET     M3020  ; S2鎖bonnet上下歸異常
7474  LDI     M624  ; 上下出,轉盤定位出
      ANI     M662  ; 上下出,轉盤定位出
      INV
      ANI     X017  ; S2鎖bonnet上下出
      OUT     T321 K3000
7481  LD      T321
      SET     M3021  ; S2鎖bonnet上下出異常
7484  LDI     M627  ; 上下歸,轉盤定位歸
      ANI     M522  ; 轉盤定位上下歸
      ANI     M665  ; 上下歸,轉盤定位歸
      INV
      ANI     X004  ; S6轉盤定位歸
      OUT     T302 K3000
7492  LD      T302
      SET     M3002  ; S6轉盤定位歸異常
7495  LDI     M624  ; 上下出,轉盤定位出
      ANI     M662  ; 上下出,轉盤定位出
      INV
      ANI     X005  ; S6轉盤定位出
      OUT     T303 K3000
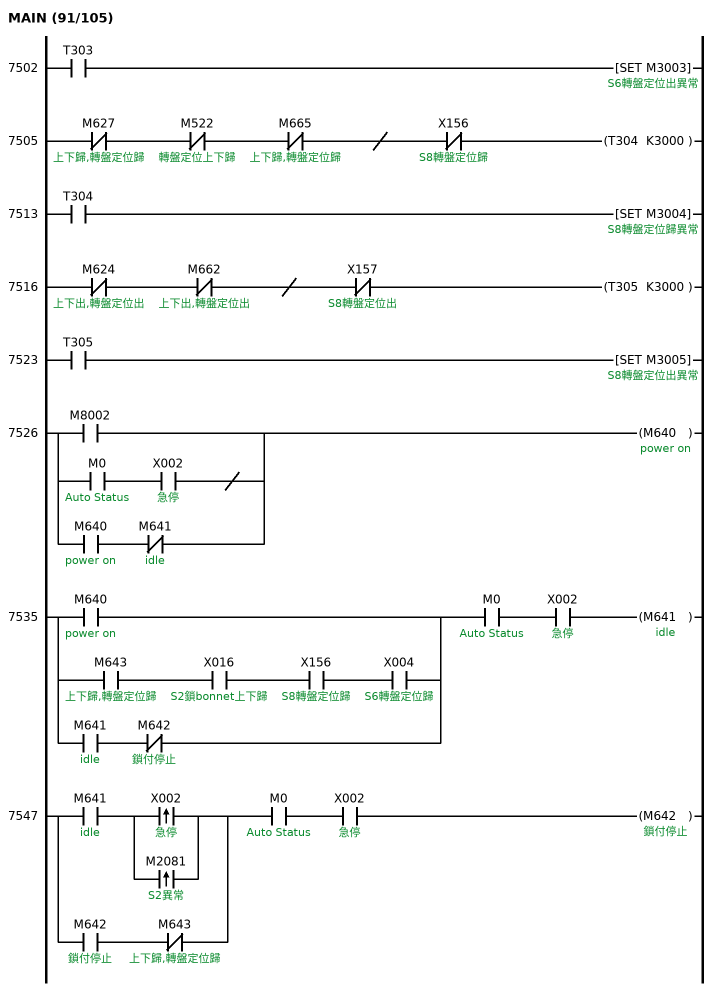
7502  LD      T303
      SET     M3003  ; S6轉盤定位出異常
7505  LDI     M627  ; 上下歸,轉盤定位歸
      ANI     M522  ; 轉盤定位上下歸
      ANI     M665  ; 上下歸,轉盤定位歸
      INV
      ANI     X156  ; S8轉盤定位歸
      OUT     T304 K3000
7513  LD      T304
      SET     M3004  ; S8轉盤定位歸異常
7516  LDI     M624  ; 上下出,轉盤定位出
      ANI     M662  ; 上下出,轉盤定位出
      INV
      ANI     X157  ; S8轉盤定位出
      OUT     T305 K3000
7523  LD      T305
      SET     M3005  ; S8轉盤定位出異常
7526  LD      M8002
      LD      M0  ; Auto Status
      AND     X002  ; 急停
      INV
      ORB
      LD      M640  ; power on
      ANI     M641  ; idle
      ORB
      OUT     M640  ; power on
7535  LD      M640  ; power on
      LD      M643  ; 上下歸,轉盤定位歸
      AND     X016  ; S2鎖bonnet上下歸
      AND     X156  ; S8轉盤定位歸
      AND     X004  ; S6轉盤定位歸
      ORB
      LD      M641  ; idle
      ANI     M642  ; 鎖付停止
      ORB
      AND     M0  ; Auto Status
      AND     X002  ; 急停
      OUT     M641  ; idle
7547  LD      M641  ; idle
      LDP     X002  ; 急停
      ORP     M2081  ; S2異常
      ANB
      LD      M642  ; 鎖付停止
      ANI     M643  ; 上下歸,轉盤定位歸
      ORB
      AND     M0  ; Auto Status
      AND     X002  ; 急停
      OUT     M642  ; 鎖付停止
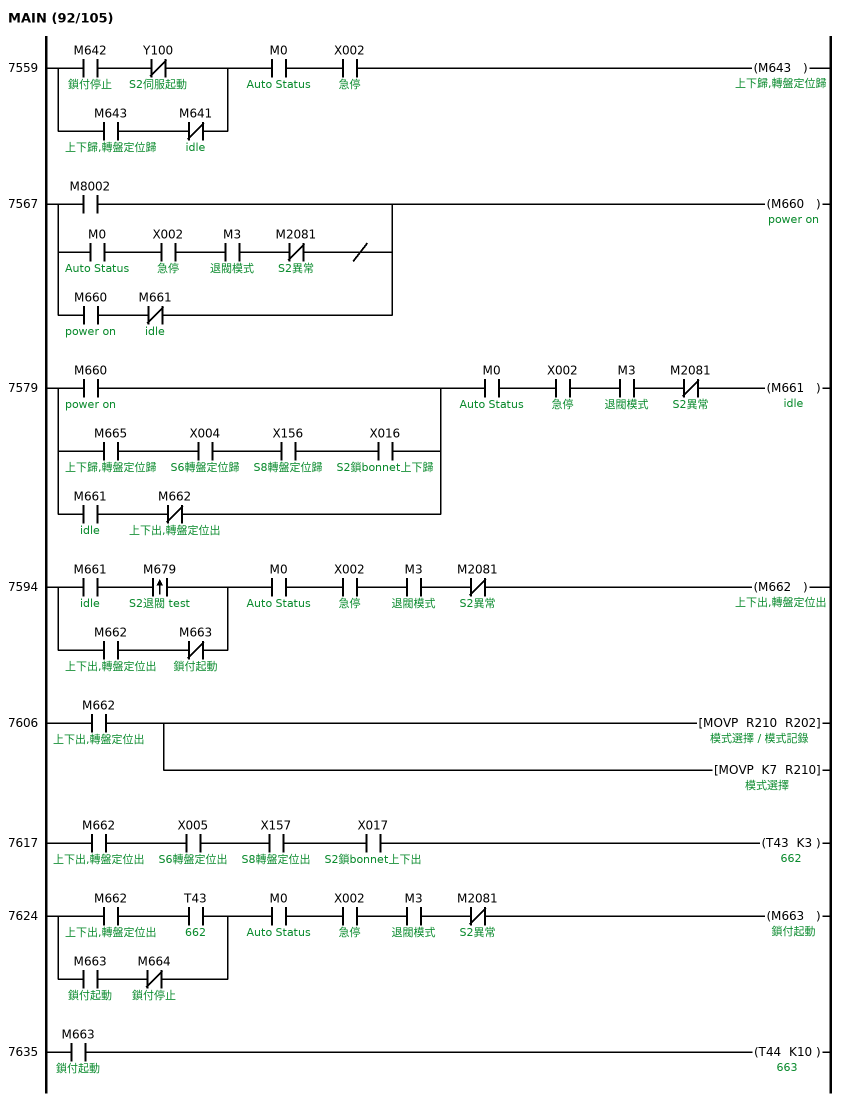
7559  LD      M642  ; 鎖付停止
      ANI     Y100  ; S2伺服起動
      LD      M643  ; 上下歸,轉盤定位歸
      ANI     M641  ; idle
      ORB
      AND     M0  ; Auto Status
      AND     X002  ; 急停
      OUT     M643  ; 上下歸,轉盤定位歸
7567  LD      M8002
      LD      M0  ; Auto Status
      AND     X002  ; 急停
      AND     M3  ; 退閥模式
      ANI     M2081  ; S2異常
      INV
      ORB
      LD      M660  ; power on
      ANI     M661  ; idle
      ORB
      OUT     M660  ; power on
7579  LD      M660  ; power on
      LD      M665  ; 上下歸,轉盤定位歸
      AND     X004  ; S6轉盤定位歸
      AND     X156  ; S8轉盤定位歸
      AND     X016  ; S2鎖bonnet上下歸
      ORB
      LD      M661  ; idle
      ANI     M662  ; 上下出,轉盤定位出
      ORB
      AND     M0  ; Auto Status
      AND     X002  ; 急停
      AND     M3  ; 退閥模式
      ANI     M2081  ; S2異常
      OUT     M661  ; idle
7594  LD      M661  ; idle
      ANDP    M679  ; S2退閥 test
      LD      M662  ; 上下出,轉盤定位出
      ANI     M663  ; 鎖付起動
      ORB
      AND     M0  ; Auto Status
      AND     X002  ; 急停
      AND     M3  ; 退閥模式
      ANI     M2081  ; S2異常
      OUT     M662  ; 上下出,轉盤定位出
7606  LD      M662  ; 上下出,轉盤定位出
      MOVP    R210 R202  ; 模式記錄
      MOVP    K7 R210
7617  LD      M662  ; 上下出,轉盤定位出
      AND     X005  ; S6轉盤定位出
      AND     X157  ; S8轉盤定位出
      AND     X017  ; S2鎖bonnet上下出
      OUT     T43 K3  ; 662
7624  LD      M662  ; 上下出,轉盤定位出
      AND     T43  ; 662
      LD      M663  ; 鎖付起動
      ANI     M664  ; 鎖付停止
      ORB
      AND     M0  ; Auto Status
      AND     X002  ; 急停
      AND     M3  ; 退閥模式
      ANI     M2081  ; S2異常
      OUT     M663  ; 鎖付起動
7635  LD      M663  ; 鎖付起動
      OUT     T44 K10  ; 663
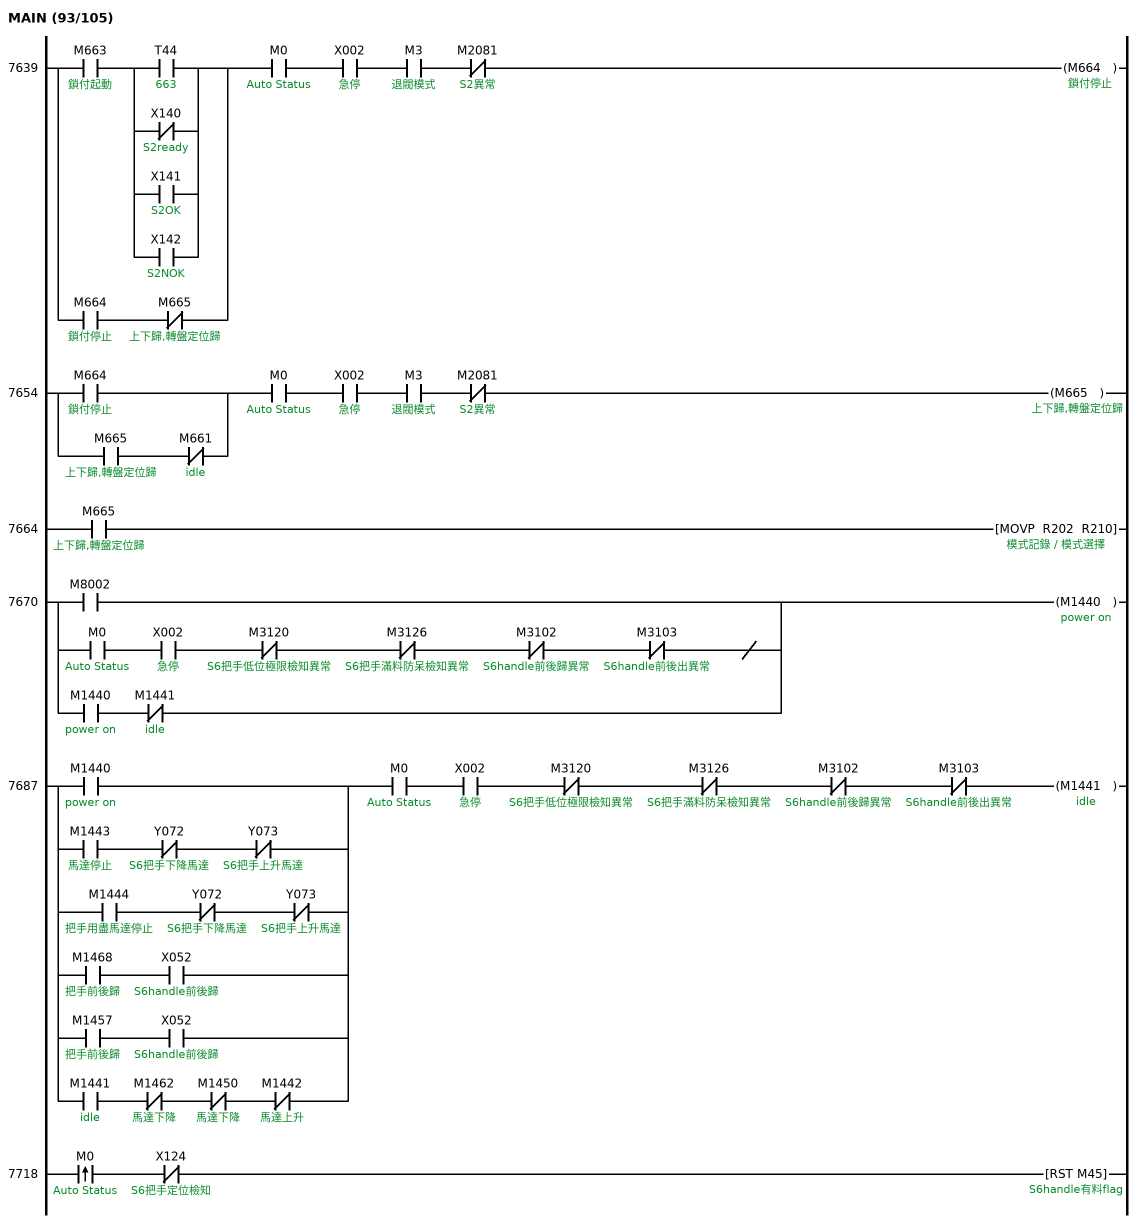
7639  LD      M663  ; 鎖付起動
      LD      T44  ; 663
      ORI     X140  ; S2ready
      OR      X141  ; S2OK
      OR      X142  ; S2NOK
      ANB
      LD      M664  ; 鎖付停止
      ANI     M665  ; 上下歸,轉盤定位歸
      ORB
      AND     M0  ; Auto Status
      AND     X002  ; 急停
      AND     M3  ; 退閥模式
      ANI     M2081  ; S2異常
      OUT     M664  ; 鎖付停止
7654  LD      M664  ; 鎖付停止
      LD      M665  ; 上下歸,轉盤定位歸
      ANI     M661  ; idle
      ORB
      AND     M0  ; Auto Status
      AND     X002  ; 急停
      AND     M3  ; 退閥模式
      ANI     M2081  ; S2異常
      OUT     M665  ; 上下歸,轉盤定位歸
7664  LD      M665  ; 上下歸,轉盤定位歸
      MOVP    R202 R210
7670  LD      M8002
      LD      M0  ; Auto Status
      AND     X002  ; 急停
      ANI     M3120  ; S6把手低位極限檢知異常
      ANI     M3126  ; S6把手滿料防呆檢知異常
      ANI     M3102  ; S6handle前後歸異常
      ANI     M3103  ; S6handle前後出異常
      INV
      ORB
      LD      M1440  ; power on
      ANI     M1441  ; idle
      ORB
      OUT     M1440  ; power on
7687  LD      M1440  ; power on
      LD      M1443  ; 馬達停止
      ANI     Y072  ; S6把手下降馬達
      ANI     Y073  ; S6把手上升馬達
      ORB
      LD      M1444  ; 把手用盡馬達停止
      ANI     Y072  ; S6把手下降馬達
      ANI     Y073  ; S6把手上升馬達
      ORB
      LD      M1468  ; 把手前後歸
      AND     X052  ; S6handle前後歸
      ORB
      LD      M1457  ; 把手前後歸
      AND     X052  ; S6handle前後歸
      ORB
      LD      M1441  ; idle
      ANI     M1462  ; 馬達下降
      ANI     M1450  ; 馬達下降
      ANI     M1442  ; 馬達上升
      ORB
      AND     M0  ; Auto Status
      AND     X002  ; 急停
      ANI     M3120  ; S6把手低位極限檢知異常
      ANI     M3126  ; S6把手滿料防呆檢知異常
      ANI     M3102  ; S6handle前後歸異常
      ANI     M3103  ; S6handle前後出異常
      OUT     M1441  ; idle
7718  LDP     M0  ; Auto Status
      ANI     X124  ; S6把手定位檢知
      RST     M45  ; S6handle有料flag
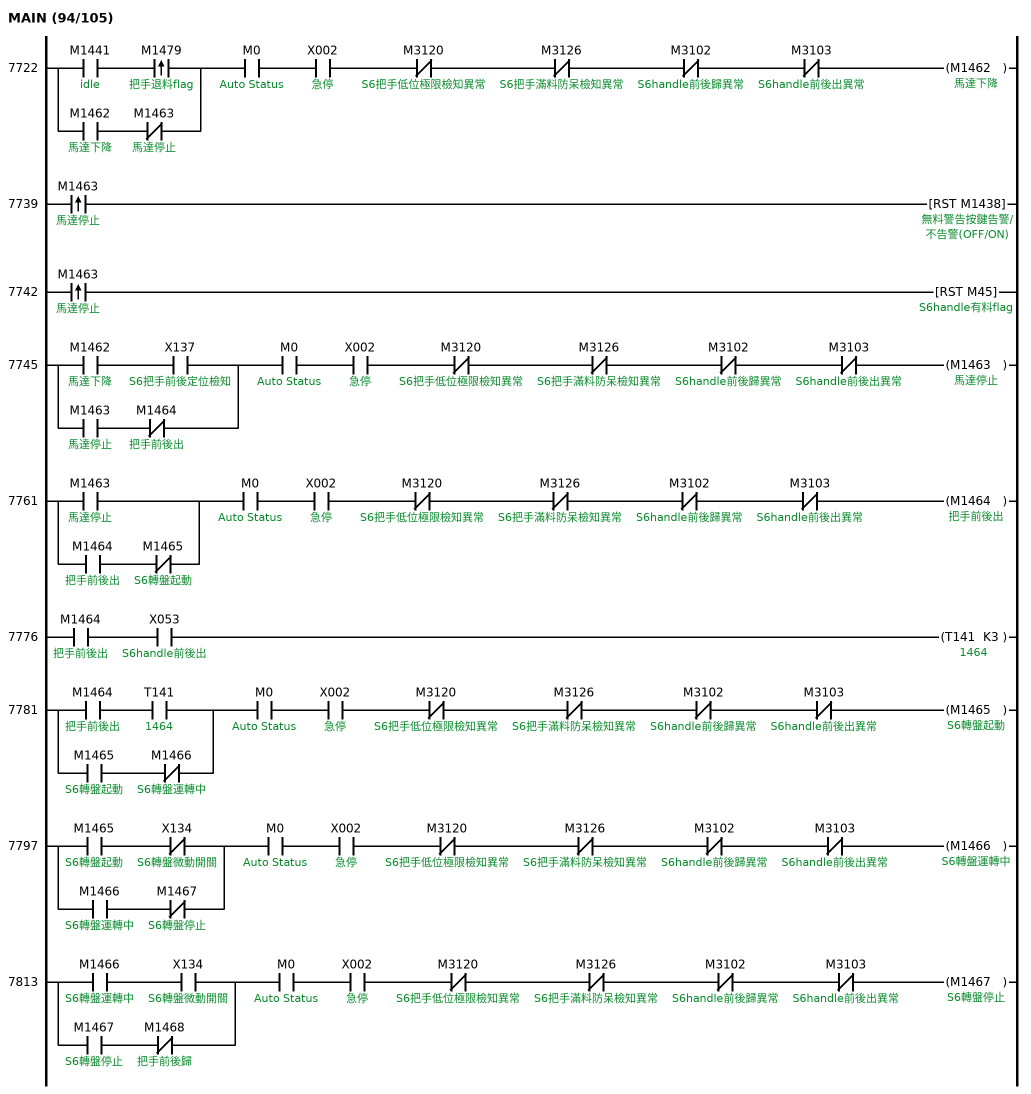
7722  LD      M1441  ; idle
      ANDP    M1479  ; 把手退料flag
      LD      M1462  ; 馬達下降
      ANI     M1463  ; 馬達停止
      ORB
      AND     M0  ; Auto Status
      AND     X002  ; 急停
      ANI     M3120  ; S6把手低位極限檢知異常
      ANI     M3126  ; S6把手滿料防呆檢知異常
      ANI     M3102  ; S6handle前後歸異常
      ANI     M3103  ; S6handle前後出異常
      OUT     M1462  ; 馬達下降
7739  LDP     M1463  ; 馬達停止
      RST     M1438  ; 無料警告按鍵告警/不告警(OFF/ON)
7742  LDP     M1463  ; 馬達停止
      RST     M45  ; S6handle有料flag
7745  LD      M1462  ; 馬達下降
      AND     X137  ; S6把手前後定位檢知
      LD      M1463  ; 馬達停止
      ANI     M1464  ; 把手前後出
      ORB
      AND     M0  ; Auto Status
      AND     X002  ; 急停
      ANI     M3120  ; S6把手低位極限檢知異常
      ANI     M3126  ; S6把手滿料防呆檢知異常
      ANI     M3102  ; S6handle前後歸異常
      ANI     M3103  ; S6handle前後出異常
      OUT     M1463  ; 馬達停止
7761  LD      M1463  ; 馬達停止
      LD      M1464  ; 把手前後出
      ANI     M1465  ; S6轉盤起動
      ORB
      AND     M0  ; Auto Status
      AND     X002  ; 急停
      ANI     M3120  ; S6把手低位極限檢知異常
      ANI     M3126  ; S6把手滿料防呆檢知異常
      ANI     M3102  ; S6handle前後歸異常
      ANI     M3103  ; S6handle前後出異常
      OUT     M1464  ; 把手前後出
7776  LD      M1464  ; 把手前後出
      AND     X053  ; S6handle前後出
      OUT     T141 K3  ; 1464
7781  LD      M1464  ; 把手前後出
      AND     T141  ; 1464
      LD      M1465  ; S6轉盤起動
      ANI     M1466  ; S6轉盤運轉中
      ORB
      AND     M0  ; Auto Status
      AND     X002  ; 急停
      ANI     M3120  ; S6把手低位極限檢知異常
      ANI     M3126  ; S6把手滿料防呆檢知異常
      ANI     M3102  ; S6handle前後歸異常
      ANI     M3103  ; S6handle前後出異常
      OUT     M1465  ; S6轉盤起動
7797  LD      M1465  ; S6轉盤起動
      ANI     X134  ; S6轉盤微動開關
      LD      M1466  ; S6轉盤運轉中
      ANI     M1467  ; S6轉盤停止
      ORB
      AND     M0  ; Auto Status
      AND     X002  ; 急停
      ANI     M3120  ; S6把手低位極限檢知異常
      ANI     M3126  ; S6把手滿料防呆檢知異常
      ANI     M3102  ; S6handle前後歸異常
      ANI     M3103  ; S6handle前後出異常
      OUT     M1466  ; S6轉盤運轉中
7813  LD      M1466  ; S6轉盤運轉中
      AND     X134  ; S6轉盤微動開關
      LD      M1467  ; S6轉盤停止
      ANI     M1468  ; 把手前後歸
      ORB
      AND     M0  ; Auto Status
      AND     X002  ; 急停
      ANI     M3120  ; S6把手低位極限檢知異常
      ANI     M3126  ; S6把手滿料防呆檢知異常
      ANI     M3102  ; S6handle前後歸異常
      ANI     M3103  ; S6handle前後出異常
      OUT     M1467  ; S6轉盤停止
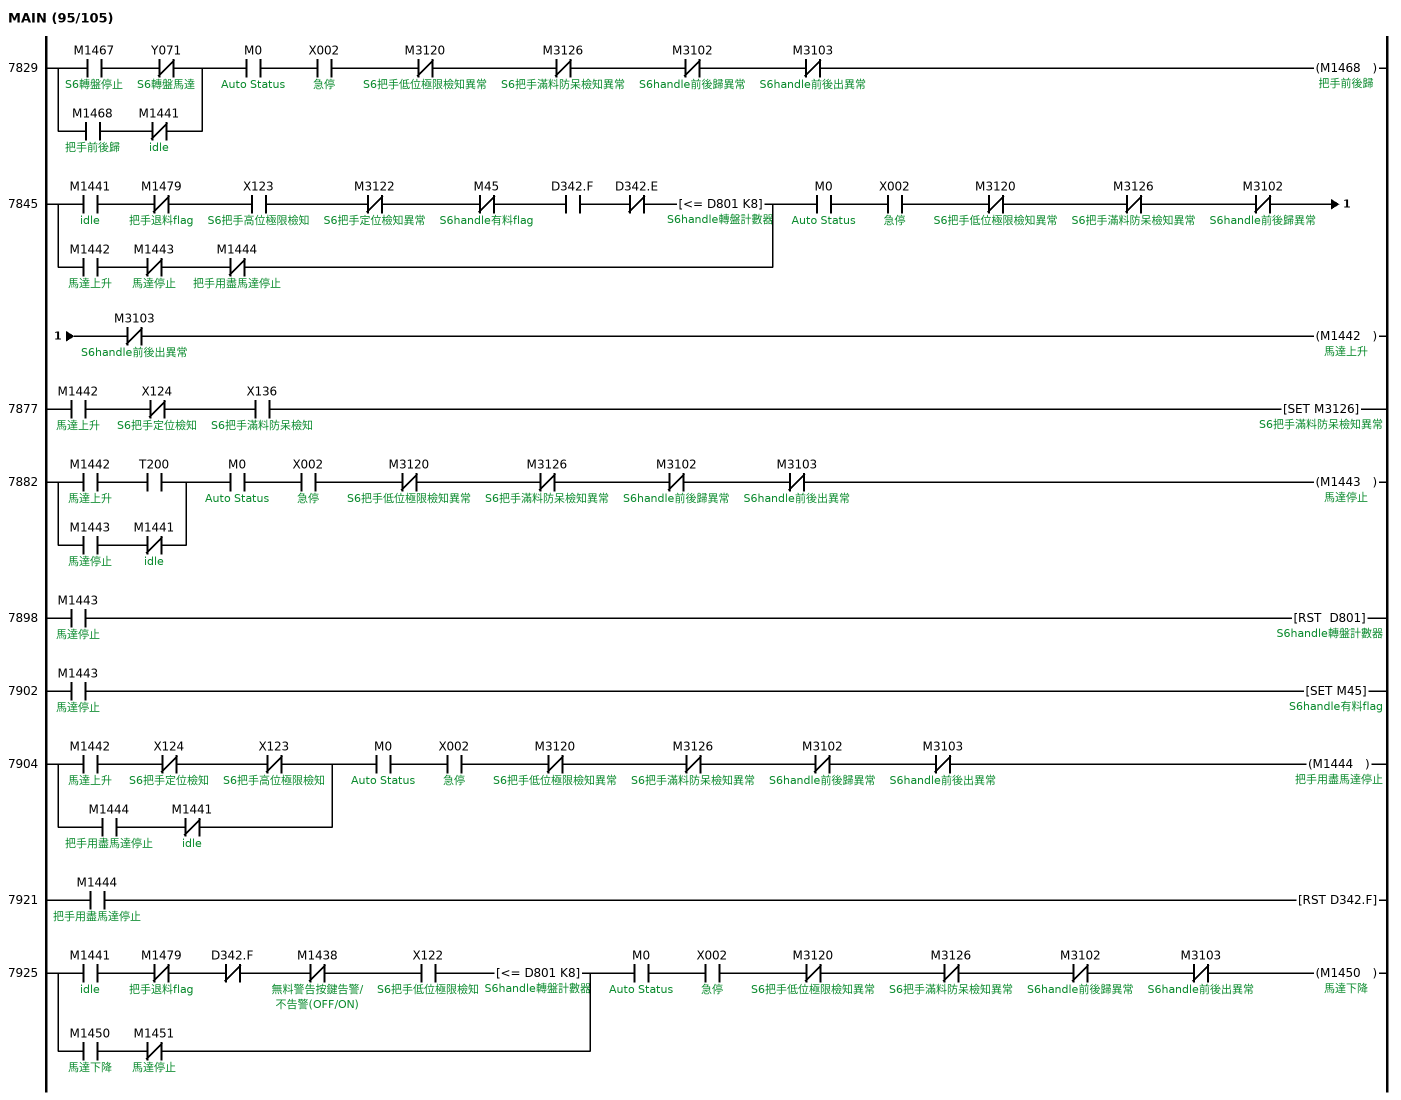
7829  LD      M1467  ; S6轉盤停止
      ANI     Y071  ; S6轉盤馬達
      LD      M1468  ; 把手前後歸
      ANI     M1441  ; idle
      ORB
      AND     M0  ; Auto Status
      AND     X002  ; 急停
      ANI     M3120  ; S6把手低位極限檢知異常
      ANI     M3126  ; S6把手滿料防呆檢知異常
      ANI     M3102  ; S6handle前後歸異常
      ANI     M3103  ; S6handle前後出異常
      OUT     M1468  ; 把手前後歸
7845  LD      M1441  ; idle
      ANI     M1479  ; 把手退料flag
      AND     X123  ; S6把手高位極限檢知
      ANI     M3122  ; S6把手定位檢知異常
      ANI     M45  ; S6handle有料flag
      AND     D342.F
      ANI     D342.E
      AND<=   D801 K8  ; S6handle轉盤計數器
      LD      M1442  ; 馬達上升
      ANI     M1443  ; 馬達停止
      ANI     M1444  ; 把手用盡馬達停止
      ORB
      AND     M0  ; Auto Status
      AND     X002  ; 急停
      ANI     M3120  ; S6把手低位極限檢知異常
      ANI     M3126  ; S6把手滿料防呆檢知異常
      ANI     M3102  ; S6handle前後歸異常
      ANI     M3103  ; S6handle前後出異常
      OUT     M1442  ; 馬達上升
7877  LD      M1442  ; 馬達上升
      ANI     X124  ; S6把手定位檢知
      AND     X136  ; S6把手滿料防呆檢知
      SET     M3126  ; S6把手滿料防呆檢知異常
7882  LD      M1442  ; 馬達上升
      AND     T200
      LD      M1443  ; 馬達停止
      ANI     M1441  ; idle
      ORB
      AND     M0  ; Auto Status
      AND     X002  ; 急停
      ANI     M3120  ; S6把手低位極限檢知異常
      ANI     M3126  ; S6把手滿料防呆檢知異常
      ANI     M3102  ; S6handle前後歸異常
      ANI     M3103  ; S6handle前後出異常
      OUT     M1443  ; 馬達停止
7898  LD      M1443  ; 馬達停止
      RST     D801  ; S6handle轉盤計數器
7902  LD      M1443  ; 馬達停止
      SET     M45  ; S6handle有料flag
7904  LD      M1442  ; 馬達上升
      ANI     X124  ; S6把手定位檢知
      ANI     X123  ; S6把手高位極限檢知
      LD      M1444  ; 把手用盡馬達停止
      ANI     M1441  ; idle
      ORB
      AND     M0  ; Auto Status
      AND     X002  ; 急停
      ANI     M3120  ; S6把手低位極限檢知異常
      ANI     M3126  ; S6把手滿料防呆檢知異常
      ANI     M3102  ; S6handle前後歸異常
      ANI     M3103  ; S6handle前後出異常
      OUT     M1444  ; 把手用盡馬達停止
7921  LD      M1444  ; 把手用盡馬達停止
      RST     D342.F
7925  LD      M1441  ; idle
      ANI     M1479  ; 把手退料flag
      ANI     D342.F
      ANI     M1438  ; 無料警告按鍵告警/不告警(OFF/ON)
      AND     X122  ; S6把手低位極限檢知
      AND<=   D801 K8  ; S6handle轉盤計數器
      LD      M1450  ; 馬達下降
      ANI     M1451  ; 馬達停止
      ORB
      AND     M0  ; Auto Status
      AND     X002  ; 急停
      ANI     M3120  ; S6把手低位極限檢知異常
      ANI     M3126  ; S6把手滿料防呆檢知異常
      ANI     M3102  ; S6handle前後歸異常
      ANI     M3103  ; S6handle前後出異常
      OUT     M1450  ; 馬達下降
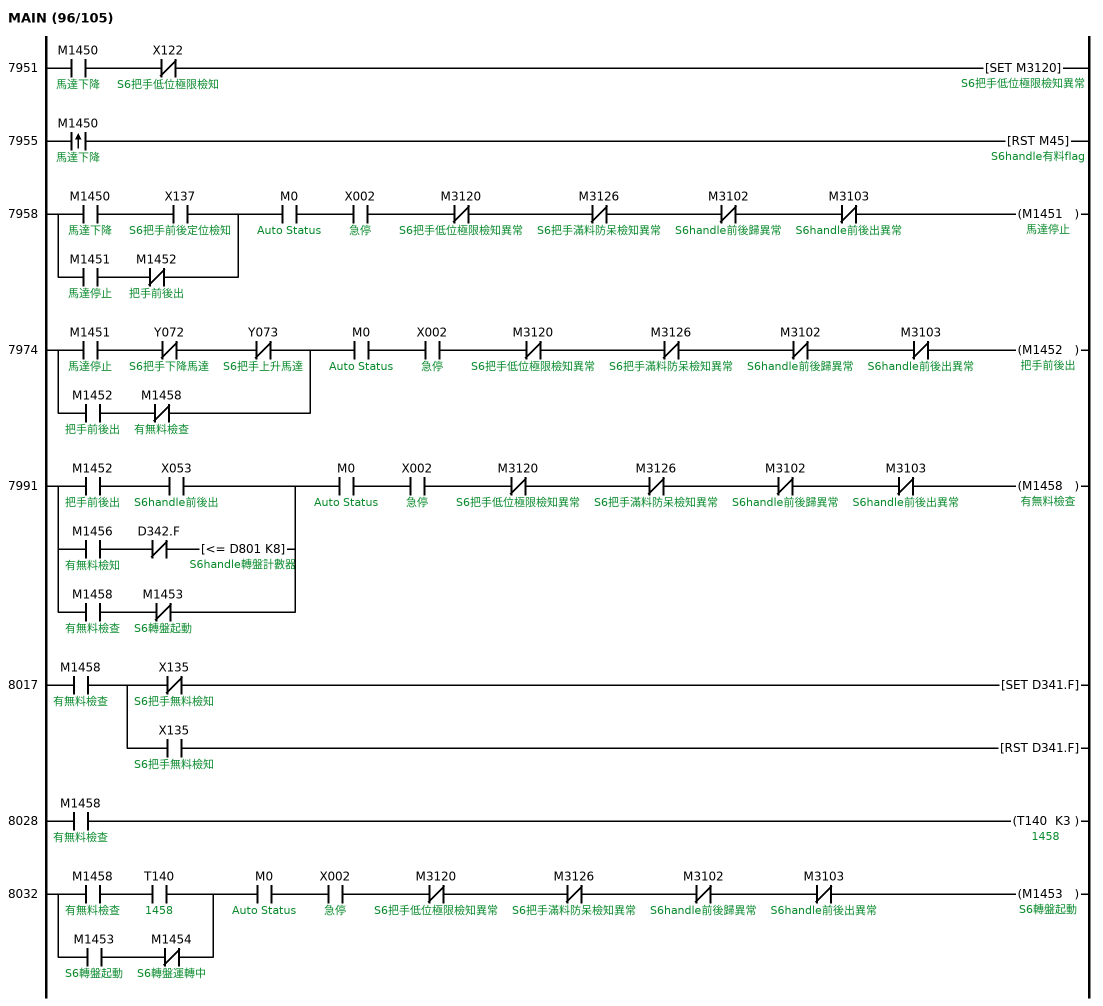
7951  LD      M1450  ; 馬達下降
      ANI     X122  ; S6把手低位極限檢知
      SET     M3120  ; S6把手低位極限檢知異常
7955  LDP     M1450  ; 馬達下降
      RST     M45  ; S6handle有料flag
7958  LD      M1450  ; 馬達下降
      AND     X137  ; S6把手前後定位檢知
      LD      M1451  ; 馬達停止
      ANI     M1452  ; 把手前後出
      ORB
      AND     M0  ; Auto Status
      AND     X002  ; 急停
      ANI     M3120  ; S6把手低位極限檢知異常
      ANI     M3126  ; S6把手滿料防呆檢知異常
      ANI     M3102  ; S6handle前後歸異常
      ANI     M3103  ; S6handle前後出異常
      OUT     M1451  ; 馬達停止
7974  LD      M1451  ; 馬達停止
      ANI     Y072  ; S6把手下降馬達
      ANI     Y073  ; S6把手上升馬達
      LD      M1452  ; 把手前後出
      ANI     M1458  ; 有無料檢查
      ORB
      AND     M0  ; Auto Status
      AND     X002  ; 急停
      ANI     M3120  ; S6把手低位極限檢知異常
      ANI     M3126  ; S6把手滿料防呆檢知異常
      ANI     M3102  ; S6handle前後歸異常
      ANI     M3103  ; S6handle前後出異常
      OUT     M1452  ; 把手前後出
7991  LD      M1452  ; 把手前後出
      AND     X053  ; S6handle前後出
      LD      M1456  ; 有無料檢知
      ANI     D342.F
      AND<=   D801 K8  ; S6handle轉盤計數器
      ORB
      LD      M1458  ; 有無料檢查
      ANI     M1453  ; S6轉盤起動
      ORB
      AND     M0  ; Auto Status
      AND     X002  ; 急停
      ANI     M3120  ; S6把手低位極限檢知異常
      ANI     M3126  ; S6把手滿料防呆檢知異常
      ANI     M3102  ; S6handle前後歸異常
      ANI     M3103  ; S6handle前後出異常
      OUT     M1458  ; 有無料檢查
8017  LD      M1458  ; 有無料檢查
      MPS
      ANI     X135  ; S6把手無料檢知
      SET     D341.F
      MPP
      AND     X135  ; S6把手無料檢知
      RST     D341.F
8028  LD      M1458  ; 有無料檢查
      OUT     T140 K3  ; 1458
8032  LD      M1458  ; 有無料檢查
      AND     T140  ; 1458
      LD      M1453  ; S6轉盤起動
      ANI     M1454  ; S6轉盤運轉中
      ORB
      AND     M0  ; Auto Status
      AND     X002  ; 急停
      ANI     M3120  ; S6把手低位極限檢知異常
      ANI     M3126  ; S6把手滿料防呆檢知異常
      ANI     M3102  ; S6handle前後歸異常
      ANI     M3103  ; S6handle前後出異常
      OUT     M1453  ; S6轉盤起動
